// TwinCAT 3 PLC project Autoloader
// ProgramVersion: 3.1.4023.0
// libraries:
//   FESTO CMMT_AS Drive Control, * (Sensata Mech Sofia)
//   Motors_AFAG_CoE, * (Sensata Technologies Bulgaria)
//   Motors_DUTs, * (Sensata Technologies Bulgaria)
//   Tc2_Math, * (Beckhoff Automation GmbH)
//   Tc2_Standard, * (Beckhoff Automation GmbH)
//   Tc2_System, * (Beckhoff Automation GmbH)
//   Tc2_TcpIp, * (Beckhoff Automation GmbH)
//   Tc2_Utilities, * (Beckhoff Automation GmbH)
//   Tc3_Module, * (Beckhoff Automation GmbH)
//   Festo_PtP_Base,3.5.10.47,Festo
//   Festo_PtP_CiA402,3.5.10.47,Festo
//   Festo_PtP_CiA402_ETC,3.5.10.47,Festo
//   Festo_PtP_CiA402_ETC_CMMT_AS,3.5.10.47,Festo
//   Festo_PtP_Virtual,3.5.10.47,Festo
//   Tc3_LinMot,1.1.0.0,NTI AG
// project tree:
//   DUTs/ camResult.TcDUT, controlCommands.TcDUT, dataRequestCam.TcDUT, dataRequestRobot.TcDUT, E_RobotStates.TcDUT, imageIO.TcDUT, ioType.TcDUT, globalDeps.TcDUT, stationBase.TcDUT
//   DUTs/Stations/incComm/ incCommDisplayStates.TcDUT, incCommImage.TcDUT, incCommIO.TcDUT, incCommSettings.TcDUT, incCommStates.TcDUT
//   DUTs/Stations/inserterLoad/ inserterLoadDisplayStates.TcDUT, inserterLoadImage.TcDUT, inserterLoadIO.TcDUT, inserterLoadRecipe.TcDUT, inserterLoadSettings.TcDUT, inserterLoadStates.TcDUT
//   DUTs/Stations/inserterUnload/ inserterUnLoadImage.TcDUT, inserterUnLoadRecipe.TcDUT, inserterUnLoadDisplayStates.TcDUT, inserterUnLoadIO.TcDUT, inserterUnLoadSettings.TcDUT, inserterUnLoadStates.TcDUT
//   DUTs/Stations/machine/ machineDisplayStates.TcDUT, machineImage.TcDUT, machineIO.TcDUT, machineSettings.TcDUT, machineStates.TcDUT
//   DUTs/Stations/roboArm/ roboArmDisplayStates.TcDUT, roboArmImage.TcDUT, roboArmIO.TcDUT, roboArmSettings.TcDUT, roboArmsRecipe.TcDUT, roboArmStates.TcDUT
//   DUTs/Stations/stackerLoad/ palletParamsL.TcDUT, stackerLoadDisplayStates.TcDUT, stackerLoadImage.TcDUT, stackerLoadIO.TcDUT, stackerLoadSettings.TcDUT, stackerLoadStates.TcDUT
//   DUTs/Stations/stackerUnload/ palletParamsU.TcDUT, stackerUnLoadDisplayStates.TcDUT, stackerUnLoadImage.TcDUT, stackerUnLoadIO.TcDUT, stackerUnLoadSettings.TcDUT, stackerUnLoadStates.TcDUT
//   GVLs/ Consts.TcGVL, DEBUG.TcGVL, Global.TcGVL, Stations.TcGVL, TagsHMI.TcGVL, TagsRobot.TcGVL
//   / PlcTask.TcTTO, RobotTask.TcTTO
//   POUs/ MAIN.TcPOU, ROBOT.TcPOU, stateMachine.TcPOU, ioControl.TcPOU
//   POUs/Mitsubishi/DUT/Communication/PacketsStructure/Input/ ST_Robot_Mitsubishi_Packet_1000.TcDUT, ST_Robot_Mitsubishi_Packet_1100.TcDUT, ST_Robot_Mitsubishi_Packet_1101.TcDUT, ST_Robot_Mitsubishi_Packet_1102.TcDUT, ST_Robot_Mitsubishi_Packet_1103.TcDUT
//   POUs/Mitsubishi/DUT/Communication/PacketsStructure/Output/ ST_Robot_Mitsubishi_Packet_2000.TcDUT, ST_Robot_Mitsubishi_Packet_2010.TcDUT, ST_Robot_Mitsubishi_Packet_2011.TcDUT, ST_Robot_Mitsubishi_Packet_2012.TcDUT, ST_Robot_Mitsubishi_Packet_2013.TcDUT, ST_Robot_Mitsubishi_Packet_2014.TcDUT, ST_Robot_Mitsubishi_Packet_2015.TcDUT, ST_Robot_Mitsubishi_Packet_2016.TcDUT, ST_Robot_Mitsubishi_Packet_2017.TcDUT, ST_Robot_Mitsubishi_Packet_2018.TcDUT, ST_Robot_Mitsubishi_Packet_2019.TcDUT, ST_Robot_Mitsubishi_Packet_2100.TcDUT, ST_Robot_Mitsubishi_Packet_2101.TcDUT
//   POUs/Mitsubishi/DUT/Communication/ ST_Robot_Misubishi_Packet_Manager.TcDUT
//   POUs/Mitsubishi/DUT/ E_Communication_Send_States.TcDUT, E_Robot_Mitsubishi_States.TcDUT, ST_Robot_Mitsubishi.TcDUT
//   POUs/Mitsubishi/ FB_Robot_Mitsubishi.TcPOU, FB_Robot_Mitsubishi_ReceivePacket.TcPOU, FB_Robot_Mitsubishi_SendPacket.TcPOU
//   POUs/Mitsubishi/Func/ FB_EXTRACT_HEX_AND_FLIP.TcPOU, FB_HEXSTR_TO_DINT.TcPOU
//   POUs/Mitsubishi/Sub/ FB_ClearOutputBuffer.TcPOU, FB_SetOutputBuffer.TcPOU
//   POUs/Stations/ incCommStation.TcPOU, insertLoadStation.TcPOU, insertUnloadStation.TcPOU, machineStation.TcPOU, roboArmStation.TcPOU, stackerLoadStation.TcPOU, stackerUnloadStation.TcPOU
// real-time tasks:
//   TASK PlcTask: cycle T#10ms, priority 20, ADS port 350
//   TASK RobotTask: cycle T#10ms, priority 1, ADS port 351
// I/O:
//   DEVICE Device 1 (EtherCAT), AmsNetId 169.254.245.124.2.1
//     Term 1 (EK1100) [EK1100 EtherCAT Coupler (2A E-Bus)]
//       Term 2 (EL1008) [EL1008 8Ch. Dig. Input 24V, 3ms]
//       Term 3 (EL1008) [EL1008 8Ch. Dig. Input 24V, 3ms]
//       Term 4 (EL1008) [EL1008 8Ch. Dig. Input 24V, 3ms]
//       Term 5 (EL2808) [EL2808 8Ch. Dig. Output 24V, 0.5A]
//       Term 6 (EL2808) [EL2808 8Ch. Dig. Output 24V, 0.5A]
//       Term 7 (EL2808) [EL2808 8Ch. Dig. Output 24V, 0.5A]
//       Term 8 (EK1310) [EK1310 EtherCAT P extension with feed-in]
//     Box 9 (EPP2316-0003) [EPP2316-0003 8 Ch. Dig. In, 10µs, 8Ch. Dig. Out 24V, 0,5A, Diagnostic, 10-Pole Plug Connector]
//     Box 10 (EPP2316-0003) [EPP2316-0003 8 Ch. Dig. In, 10µs, 8Ch. Dig. Out 24V, 0,5A, Diagnostic, 10-Pole Plug Connector]
//     Box 11 (CMMT-AS) [CMMT-AS]
//     Box 12 (CMMT-AS) [CMMT-AS]
//     Box 13 (C1150-EC-XC-1S) [C1150-EC-XC-1S V1.7b5]
//     Box 14 (C1150-EC-XC-1S) [C1150-EC-XC-1S V1.7b5]
//     Box 15 (EX260-SEC1) [EX260-SEC1 EtherCAT SI Unit (32DO_PNP) Rev1.2]
//     Box 16 (EP1008-0001) [EP1008-0001 8 Ch. Dig. Input 24V, 3ms, M8]
//     Box 17 (EP1008-0001) [EP1008-0001 8 Ch. Dig. Input 24V, 3ms, M8]
//     Box 18 (EP1008-0001) [EP1008-0001 8 Ch. Dig. Input 24V, 3ms, M8]
// variable links:
//   Autoloader/Autoloader Instance <-> Device 1 (EtherCAT)/Box 10 (EPP2316-0003)
//     PlcTask Inputs/Global.INPUT_IMAGE[10] <-> DIG Inputs/Input 1
//     PlcTask Inputs/Global.INPUT_IMAGE[10] @bit {1..7} <-> DIG Inputs/Input {2..8}  (7 links)
//     PlcTask Outputs/Global.OUTPUT_IMAGE[10] <-> DIG Outputs/Output 1
//     PlcTask Outputs/Global.OUTPUT_IMAGE[10] @bit {1..7} <-> DIG Outputs/Output {2..8}  (7 links)
//   Autoloader/Autoloader Instance <-> Device 1 (EtherCAT)/Box 11 (CMMT-AS)
//     PlcTask Inputs/Stations.sLoadAxis.AdsAddr_In <-> InfoData/AdsAddr
//     PlcTask Inputs/Stations.sLoadAxis.ModesOfOperationDisplay_In <-> Inputs/Modes of operation display
//     PlcTask Inputs/Stations.sLoadAxis.PositionActualValue_In <-> Inputs/Position actual value
//     PlcTask Inputs/Stations.sLoadAxis.SlaveState_In <-> InfoData/State
//     PlcTask Inputs/Stations.sLoadAxis.Statusword_In <-> Inputs/Statusword
//     PlcTask Inputs/Stations.sLoadAxis.TorqueActualValue_In <-> Inputs/Torque actual value
//     PlcTask Inputs/Stations.sLoadAxis.VelocityActualValue_In <-> Inputs/Velocity actual value
//     PlcTask Inputs/Stations.sLoadAxis.WcState_In <-> WcState/WcState
//     PlcTask Outputs/Stations.sLoadAxis.Controlword_Out <-> Outputs/Controlword
//     PlcTask Outputs/Stations.sLoadAxis.ModesOfOperation_Out <-> Outputs/Modes of operation
//     PlcTask Outputs/Stations.sLoadAxis.ProfileVelocity_Out <-> Outputs/Profile velocity
//     PlcTask Outputs/Stations.sLoadAxis.TargetPosition_Out <-> Outputs/Target position
//     PlcTask Outputs/Stations.sLoadAxis.TargetTorque_Out <-> Outputs/Target torque
//     PlcTask Outputs/Stations.sLoadAxis.TargetVelocity_Out <-> Outputs/Target velocity
//   Autoloader/Autoloader Instance <-> Device 1 (EtherCAT)/Box 12 (CMMT-AS)
//     PlcTask Inputs/Stations.sUnloadAxis.AdsAddr_In <-> InfoData/AdsAddr
//     PlcTask Inputs/Stations.sUnloadAxis.ModesOfOperationDisplay_In <-> Inputs/Modes of operation display
//     PlcTask Inputs/Stations.sUnloadAxis.PositionActualValue_In <-> Inputs/Position actual value
//     PlcTask Inputs/Stations.sUnloadAxis.SlaveState_In <-> InfoData/State
//     PlcTask Inputs/Stations.sUnloadAxis.Statusword_In <-> Inputs/Statusword
//     PlcTask Inputs/Stations.sUnloadAxis.TorqueActualValue_In <-> Inputs/Torque actual value
//     PlcTask Inputs/Stations.sUnloadAxis.VelocityActualValue_In <-> Inputs/Velocity actual value
//     PlcTask Inputs/Stations.sUnloadAxis.WcState_In <-> WcState/WcState
//     PlcTask Outputs/Stations.sUnloadAxis.Controlword_Out <-> Outputs/Controlword
//     PlcTask Outputs/Stations.sUnloadAxis.ModesOfOperation_Out <-> Outputs/Modes of operation
//     PlcTask Outputs/Stations.sUnloadAxis.ProfileVelocity_Out <-> Outputs/Profile velocity
//     PlcTask Outputs/Stations.sUnloadAxis.TargetPosition_Out <-> Outputs/Target position
//     PlcTask Outputs/Stations.sUnloadAxis.TargetTorque_Out <-> Outputs/Target torque
//     PlcTask Outputs/Stations.sUnloadAxis.TargetVelocity_Out <-> Outputs/Target velocity
//   Autoloader/Autoloader Instance <-> Device 1 (EtherCAT)/Box 13 (C1150-EC-XC-1S)
//     PlcTask Inputs/Stations.insertLoadAxis.DrvToPlc/ComActualPosition <-> Default Inputs/ActualPosition
//     PlcTask Inputs/Stations.insertLoadAxis.DrvToPlc/ComDemandPosition <-> Default Inputs/DemandPosition
//     PlcTask Inputs/Stations.insertLoadAxis.DrvToPlc/StateVar <-> Default Inputs/StateVar
//     PlcTask Inputs/Stations.insertLoadAxis.DrvToPlc/StatusWord <-> Default Inputs/StatusWord
//     PlcTask Inputs/Stations.insertLoadAxis.DrvToPlc/WarnWord <-> Default Inputs/WarnWord
//     PlcTask Outputs/Stations.insertLoadAxis.PlcToDrv/ControlWord <-> Default Outputs/Control Word
//     PlcTask Outputs/Stations.insertLoadAxis.PlcToDrv/MCHeader <-> Default Outputs/Motion Command Header
//     PlcTask Outputs/Stations.insertLoadAxis.PlcToDrv/MCParaDWord_00_03 <-> Default Outputs/Motion Command Par 1
//     PlcTask Outputs/Stations.insertLoadAxis.PlcToDrv/MCParaDWord_04_07 <-> Default Outputs/Motion Command Par 2
//     PlcTask Outputs/Stations.insertLoadAxis.PlcToDrv/MCParaDWord_08_11 <-> Default Outputs/Motion Command Par 3
//     PlcTask Outputs/Stations.insertLoadAxis.PlcToDrv/MCParaDWord_12_15 <-> Default Outputs/Motion Command Par 4
//     PlcTask Outputs/Stations.insertLoadAxis.PlcToDrv/MCParaDWord_16_19 <-> Default Outputs/Motion Command Par 5
//   Autoloader/Autoloader Instance <-> Device 1 (EtherCAT)/Box 14 (C1150-EC-XC-1S)
//     PlcTask Inputs/Stations.insertUnLoadAxis.DrvToPlc/ComActualPosition <-> Default Inputs/ActualPosition
//     PlcTask Inputs/Stations.insertUnLoadAxis.DrvToPlc/ComDemandPosition <-> Default Inputs/DemandPosition
//     PlcTask Inputs/Stations.insertUnLoadAxis.DrvToPlc/StateVar <-> Default Inputs/StateVar
//     PlcTask Inputs/Stations.insertUnLoadAxis.DrvToPlc/StatusWord <-> Default Inputs/StatusWord
//     PlcTask Inputs/Stations.insertUnLoadAxis.DrvToPlc/WarnWord <-> Default Inputs/WarnWord
//     PlcTask Outputs/Stations.insertUnLoadAxis.PlcToDrv/ControlWord <-> Default Outputs/Control Word
//     PlcTask Outputs/Stations.insertUnLoadAxis.PlcToDrv/MCHeader <-> Default Outputs/Motion Command Header
//     PlcTask Outputs/Stations.insertUnLoadAxis.PlcToDrv/MCParaDWord_00_03 <-> Default Outputs/Motion Command Par 1
//     PlcTask Outputs/Stations.insertUnLoadAxis.PlcToDrv/MCParaDWord_04_07 <-> Default Outputs/Motion Command Par 2
//     PlcTask Outputs/Stations.insertUnLoadAxis.PlcToDrv/MCParaDWord_08_11 <-> Default Outputs/Motion Command Par 3
//     PlcTask Outputs/Stations.insertUnLoadAxis.PlcToDrv/MCParaDWord_12_15 <-> Default Outputs/Motion Command Par 4
//     PlcTask Outputs/Stations.insertUnLoadAxis.PlcToDrv/MCParaDWord_16_19 <-> Default Outputs/Motion Command Par 5
//   Autoloader/Autoloader Instance <-> Device 1 (EtherCAT)/Box 15 (EX260-SEC1)
//     PlcTask Outputs/Global.OUTPUT_IMAGE[150] <-> Byte 0/Output
//     PlcTask Outputs/Global.OUTPUT_IMAGE[151] <-> Byte 1/Output
//     PlcTask Outputs/Global.OUTPUT_IMAGE[152] <-> Byte 2/Output
//   Autoloader/Autoloader Instance <-> Device 1 (EtherCAT)/Box 16 (EP1008-0001)
//     PlcTask Inputs/Global.INPUT_IMAGE[16] <-> Channel 1/Input
//     PlcTask Inputs/Global.INPUT_IMAGE[16] @bit {1..7} <-> Channel {2..8}/Input  (7 links)
//   Autoloader/Autoloader Instance <-> Device 1 (EtherCAT)/Box 17 (EP1008-0001)
//     PlcTask Inputs/Global.INPUT_IMAGE[17] <-> Channel 1/Input
//     PlcTask Inputs/Global.INPUT_IMAGE[17] @bit {1..7} <-> Channel {2..8}/Input  (7 links)
//   Autoloader/Autoloader Instance <-> Device 1 (EtherCAT)/Box 18 (EP1008-0001)
//     PlcTask Inputs/Global.INPUT_IMAGE[18] <-> Channel 1/Input
//     PlcTask Inputs/Global.INPUT_IMAGE[18] @bit {1..7} <-> Channel {2..8}/Input  (7 links)
//   Autoloader/Autoloader Instance <-> Device 1 (EtherCAT)/Box 9 (EPP2316-0003)
//     PlcTask Inputs/Global.INPUT_IMAGE[9] <-> DIG Inputs/Input 1
//     PlcTask Inputs/Global.INPUT_IMAGE[9] @bit {1..7} <-> DIG Inputs/Input {2..8}  (7 links)
//     PlcTask Outputs/Global.OUTPUT_IMAGE[9] <-> DIG Outputs/Output 1
//     PlcTask Outputs/Global.OUTPUT_IMAGE[9] @bit {1..7} <-> DIG Outputs/Output {2..8}  (7 links)
//   Autoloader/Autoloader Instance <-> Device 1 (EtherCAT)/Term 1 (EK1100)/Term 2 (EL1008)
//     PlcTask Inputs/Global.INPUT_IMAGE[2] <-> Channel 1/Input
//     PlcTask Inputs/Global.INPUT_IMAGE[2] @bit {1..7} <-> Channel {2..8}/Input  (7 links)
//   Autoloader/Autoloader Instance <-> Device 1 (EtherCAT)/Term 1 (EK1100)/Term 3 (EL1008)
//     PlcTask Inputs/Global.INPUT_IMAGE[3] <-> Channel 1/Input
//     PlcTask Inputs/Global.INPUT_IMAGE[3] @bit {1..7} <-> Channel {2..8}/Input  (7 links)
//   Autoloader/Autoloader Instance <-> Device 1 (EtherCAT)/Term 1 (EK1100)/Term 4 (EL1008)
//     PlcTask Inputs/Global.INPUT_IMAGE[4] <-> Channel 1/Input
//     PlcTask Inputs/Global.INPUT_IMAGE[4] @bit {1..7} <-> Channel {2..8}/Input  (7 links)
//   Autoloader/Autoloader Instance <-> Device 1 (EtherCAT)/Term 1 (EK1100)/Term 5 (EL2808)
//     PlcTask Outputs/Global.OUTPUT_IMAGE[5] <-> Channel 1/Output
//     PlcTask Outputs/Global.OUTPUT_IMAGE[5] @bit {1..7} <-> Channel {2..8}/Output  (7 links)
//   Autoloader/Autoloader Instance <-> Device 1 (EtherCAT)/Term 1 (EK1100)/Term 6 (EL2808)
//     PlcTask Outputs/Global.OUTPUT_IMAGE[6] <-> Channel 1/Output
//     PlcTask Outputs/Global.OUTPUT_IMAGE[6] @bit {1..7} <-> Channel {2..8}/Output  (7 links)
//   Autoloader/Autoloader Instance <-> Device 1 (EtherCAT)/Term 1 (EK1100)/Term 7 (EL2808)
//     PlcTask Outputs/Global.OUTPUT_IMAGE[7] <-> Channel 1/Output
//     PlcTask Outputs/Global.OUTPUT_IMAGE[7] @bit {1..7} <-> Channel {2..8}/Output  (7 links)

CONFIGURATION Autoloader
    RESOURCE PLC ON TwinCAT3
        TASK PlcTask(INTERVAL := T#10ms, PRIORITY := 20);
        TASK RobotTask(INTERVAL := T#10ms, PRIORITY := 1);
        PROGRAM MAIN WITH PlcTask : MAIN;
        PROGRAM Robot WITH RobotTask : Robot;
    END_RESOURCE
END_CONFIGURATION

// ---- DUTs/camResult.TcDUT
{attribute 'qualified_only'}

TYPE camResult :
(
	null          := 0,                         // Неправилен резултат от камерата
	turnCCW,
	turnCW
	
)DINT;
END_TYPE

// ---- DUTs/controlCommands.TcDUT
{attribute 'qualified_only'}

// Команди който идват от I&C

TYPE controlCommands :
(
	null		:= 0,
	stop,
	start
	
)DINT;
END_TYPE

// ---- DUTs/dataRequestCam.TcDUT
{attribute 'qualified_only'}




TYPE dataRequestCam :
(
	done               := Consts.NO_REQUEST,
	error              := Consts.REQUEST_ERROR,
	
	camShotRecipe1     := 1,           // Тази стойност НЕ трябва да се променя - винаги е 1 !
	camShotRecipe2,
	camShotRecipe3,
	camShotRecipe4,
	camShotRecipe5,
	camShotRecipe6,
	camShotRecipe7,
	camShotRecipe8,
	camShotRecipe9,
	camShotRecipe10,
	camShotRecipe11,
	camShotRecipe12,
	camShotRecipe13,
	camShotRecipe14,
	camShotRecipe15
	
	
)DINT;
END_TYPE

// ---- DUTs/dataRequestRobot.TcDUT
{attribute 'qualified_only'}


TYPE dataRequestRobot :
(
	

	done       := Consts.NO_REQUEST,
	error      := Consts.REQUEST_ERROR,
	
	roboInit	   := 100,				// Зарежда MAINPROGRAM и изчаква робота да е в READY
	
	roboPrg_Home   := 1,
	roboPrg_SensorLoad,
	roboPrg_SensorUnload,
	roboPrg_SensorDown,
	roboPrg_PreLoad,
	roboPrg_Load,
	roboPrg_PreUnload,
	roboPrg_Unload,
	roboPrg_LoadStacker,
	roboPrg_UnloadStacker,
	roboPrg_EmptyPlace,
	roboPrg_HomeWithPallet
	
)DINT;
END_TYPE

// ---- DUTs/E_RobotStates.TcDUT
{attribute 'qualified_only'}
{attribute 'to_string'}
TYPE E_RobotStates :
(
	STATE_WAITING_FOR_INIT := 0,
	STATE_INIT_ROBOT_TOGGLE,
	STATE_INIT_ROBOT_ON,
	STATE_INIT_CHECK_ROBOT_ERROR,
	STATE_INIT_CHECK_ROBOT_ERROR_DONE,
	STATE_INIT_CHECK_ROBOT_READY,
	STATE_INIT_CHECK_ROBOT_READY_DONE,
	STATE_INIT_CHECK_ROBOT_SERVOON,
	STATE_INIT_CHECK_ROBOT_SERVOON_DONE,
	STATE_INIT_DONE,
	STATE_WAITING_FOR_COMMAND := 100,
	STATE_WAITING_START_PRG,
	STATE_PROGRAM_DONE,	//Ready
	STATE_ERROR := 1000	// Default error
) UDINT;
END_TYPE

// ---- DUTs/imageIO.TcDUT
TYPE imageIO :
STRUCT
	
	// Това е структура която "вързва" даден сигнал от stataionIO с опеделен такъв от В/И image на TC
	// Идеята е да не се мисли за обновяване на сигналите, т.е. да няма копиране на няколко места за да се обнови статуса им.
	// TO DO -> да се реализира подхода и за аналогови сигнали 
	
	stIO			: REFERENCE TO BOOL; 						                // име на сигнал от stationIO
	image			: POINTER TO ARRAY [0..Consts.MAX_IO_POINTS] OF BYTE;       // масив на IO image
	iType           : ioType; 													// тип
	iByte 			: UINT;                                                     // номер на байт от масива
	iBit			: UINT; 									                // номер на бит от байта
	 
END_STRUCT
END_TYPE

// ---- DUTs/ioType.TcDUT
{attribute 'qualified_only'}

// Опеределя вида на перифериятя - за сега е само входе и изходен бит

TYPE ioType :
(
	INPUT_BIT   := 1,
	OUTPUT_BIT
)DINT;
END_TYPE

// ---- DUTs/globalDeps.TcDUT
{attribute 'qualified_only'}

TYPE globalDeps :
(
	
	// За machine station
	depMachineInitDone 			:=    10,
	depMachineAuto,
	depMachineStopping, 
	depMachineStop,
	depMachinePurgeStart,
	depMachinePurgeRobot,
	depMacinePurgeStackers,

	// За staker load station
	depSLoadInit,
	depSLoadWaitRobotReady,
	depSLoadRobotOutOfReach,
	depSLoadStop,
	depSLoadPurgeDone,
	depSLoadRobotLoadGrip,
	depSLoadStationReady,
	depSLoadStationDone,
	
	// За staker unload station
	depSUnloadInit,
	depSUnloadStop,
	depSUnloadWaitRobotReady,
	depSUnloadRobotUnloadGrip,
	depSUnloadRobotOutOfReach,	
	depSUnloadPurgeDone,
	depSUnloadStationReady,
	
	// За Inc Comm station
	depIncCommModeDone,
	depIncIncComm,
	depIncCycleDone,
	depIncStop,
	depIncPurgeDone,
	
	// За RoboArm station
	depRoboInitDone,
	depRoboStop,
	depRoboLoadPalletUnlock,
	depRoboUnLoadPalletLock,
	depRoboUnLodPalletFull,
	depRoboPurgeDone,
	depRoboGripOpen,
	depRoboGripClose,
	depRoboILoadOnPos,
	depRoboULoadOnPos,
	depRoboLoadSensor,
	depRoboStartLoadStacker,
	depRobotClearUnLoadStacker,
	
	// За inserter load station
	depILoadInitDone,
    depILoadWaitRobotReady,	
	depILoadRobotBack,
	depILoadSignalForLoad,
	depILoadWaitIndex,
	depILoadDone,
	depILoadStop,
	
	// За inserter unload station
	depULoadInitDone,
    depULoadWaitRobotReady,	
	depULoadWaitIndex,
	depULoadDone,
	depULoadRobotOutOfRich,	
	depULoadStop
	
)DINT;
END_TYPE

// ---- DUTs/Stations/incComm/incCommDisplayStates.TcDUT
{attribute 'qualified_only'}

TYPE incCommDisplayStates :
(
	
	dStStartingUp   := 10,
	dStStandBy,
	dStIncModeSignalsError,
	dStWaitForAllStatinsReady,
	dStDialTableIndexPermition,
	dStDialTableIndexReady,
	dStStationIsStopped,
	dStWaitForNextStep
	
	
	
)DINT;
END_TYPE

// ---- DUTs/Stations/incComm/incCommImage.TcDUT
TYPE incCommImage :
STRUCT
	
	// Входове
    xSignalStop 		: imageIO := ( stIO   := Stations.incCommHmiIO.x_SignalStop,
									   image  := ADR(Global.INPUT_IMAGE),
									   iType  := ioType.INPUT_BIT,
									   iByte  := 4,
									   iBit   := 0 );	
									   
    xSignalStart 		: imageIO := ( stIO   := Stations.incCommHmiIO.x_SignalStart,
									   image  := ADR(Global.INPUT_IMAGE),
									   iType  := ioType.INPUT_BIT,
									   iByte  := 4,
									   iBit   := 1 );

    xPickNestLoaded 	: imageIO := ( stIO   := Stations.incCommHmiIO.x_pickNestLoaded,
									   image  := ADR(Global.INPUT_IMAGE),
									   iType  := ioType.INPUT_BIT,
									   iByte  := 4,
									   iBit   := 2 );
									   
    xDailIndexDone 	: imageIO := ( stIO   := Stations.incCommHmiIO.x_DailIndexDone,
									   image  := ADR(Global.INPUT_IMAGE),
									   iType  := ioType.INPUT_BIT,
									   iByte  := 4,
									   iBit   := 3);									   

    xRecipeBit0 	    : imageIO := ( stIO   := Stations.incCommHmiIO.x_recipeBit0,
									   image  := ADR(Global.INPUT_IMAGE),
									   iType  := ioType.INPUT_BIT,
									   iByte  := 4,
									   iBit   := 4);

    xRecipeBit1 	    : imageIO := ( stIO   := Stations.incCommHmiIO.x_recipeBit1,
									   image  := ADR(Global.INPUT_IMAGE),
									   iType  := ioType.INPUT_BIT,
									   iByte  := 4,
									   iBit   := 5);	
									   
   xRecipeBit2 	    	: imageIO := ( stIO   := Stations.incCommHmiIO.x_recipeBit2,
									   image  := ADR(Global.INPUT_IMAGE),
									   iType  := ioType.INPUT_BIT,
									   iByte  := 4,
									   iBit   := 6);

   xRecipeBit3 	    	: imageIO := ( stIO   := Stations.incCommHmiIO.x_recipeBit3,
									   image  := ADR(Global.INPUT_IMAGE),
									   iType  := ioType.INPUT_BIT,
									   iByte  := 4,
									   iBit   := 7);									   
									   									   

	// Изходи
    yProductChange 		: imageIO := ( stIO   := Stations.incCommHmiIO.y_productChange,
									   image  := ADR(Global.OUTPUT_IMAGE),
									   iType  := ioType.OUTPUT_BIT,
									   iByte  := 5,
									   iBit   := 0 );

    yAlarm 		        : imageIO := ( stIO   := Stations.incCommHmiIO.y_alarm,
									   image  := ADR(Global.OUTPUT_IMAGE),
									   iType  := ioType.OUTPUT_BIT,
									   iByte  := 5,
									   iBit   := 1 );

    yDailIndex 		    : imageIO := ( stIO   := Stations.incCommHmiIO.y_dailIndex,
									   image  := ADR(Global.OUTPUT_IMAGE),
									   iType  := ioType.OUTPUT_BIT,
									   iByte  := 5,
									   iBit   := 2 );	
					   	

END_STRUCT
END_TYPE

// ---- DUTs/Stations/incComm/incCommIO.TcDUT
TYPE incCommIO :
STRUCT
	
	// Входове
	x_SignalStop			: BOOL; 						// Стоп бутон на InC
	x_SignalStart			: BOOL; 						// Старт бутон на InC
	x_pickNestLoaded        : BOOL; 						// Има готова бройка за взимане 						// Може да се остави бройка - гнездото е празно
	x_recipeBit0			: BOOL; 						// Режим на работа HEX24
    x_recipeBit1			: BOOL;							// Режим на работа HEX27
	x_recipeBit2            : BOOL;
	x_recipeBit3            : BOOL;
	x_dailIndexDone			: BOOL;							// Индекс масата е направила един ход - движението е завършено       
	
	// Изходи
	y_productChange			: BOOL;                         // InC има разрешение да стартира нов лот (и да смени продукта HEX24 или HEX27)
	y_alarm					: BOOL; 						// Има активна аларма
	y_dailIndex				: BOOL; 						// InC е безопастно да завърти индекс масата с един ход

END_STRUCT
END_TYPE

// ---- DUTs/Stations/incComm/incCommSettings.TcDUT
TYPE incCommSettings :
STRUCT
END_STRUCT
END_TYPE

// ---- DUTs/Stations/incComm/incCommStates.TcDUT
{attribute 'qualified_only'}

TYPE incCommStates :
(
		stNull      :=    Consts.ST_NULL,
		stStartUp   :=    Consts.ST_START_UP,
		stInit      :=    Consts.ST_INIT,
		stReady     :=    Consts.ST_READY,
		stStop      :=    Consts.ST_STOP,
		stStepBlock :=    Consts.ST_STEP_BLOCK,	
		stEMG		:=    Consts.ST_EMG,
		
		
		stSetMode                := 1000,
		stStationStop,
		
		stIndexStart,
		stIndexEnableStations,
		stIndexStationsReady,
		stSignalStations,		
		stIndexEnable, 
		stIndexReady,
		stIndexCheck, 
		stIndexDone,
		
		stPurgeStart,
		stPurgeFinish,
		stPurgeDone,

		stErrCommFault

)DINT;
END_TYPE

// ---- DUTs/Stations/inserterLoad/inserterLoadDisplayStates.TcDUT
{attribute 'qualified_only'}

TYPE inserterLoadDisplayStates :
(
	
	dStStartUp,
	dStStandBy,
	dStStationIsStopped,
	dStStationIsReseting,
	dStWorking,
	dStStationReady,
	dStWaitForNextStep,
	
	dStGripperDidNotClose,
	dStGripperDidNotOpen,
	dStInserterDidNotMoveDown,
	dStInserterDidNotMoveUp,
	dStDriveDidNotHome,
	dStDriveTimeOutMove,
	dStDriveError,
	dStCameraTimeOut,
	dStCameraError,
	dStCameraBadResult,
	dStInitSensorGripError
	
	
)DINT;
END_TYPE

// ---- DUTs/Stations/inserterLoad/inserterLoadImage.TcDUT
TYPE inserterLoadImage :
STRUCT
	
   // Входове
   xGrip_open 	        : imageIO := ( stIO   := Stations.insertLoadHmiIO.x_Grip_open,
									   image  := ADR(Global.INPUT_IMAGE),
									   iType  := ioType.INPUT_BIT,
									   iByte  := 18,
									   iBit   := 0 );	
									   
   xGrip_close			: imageIO := ( stIO   := Stations.insertLoadHmiIO.x_Grip_close,
									   image  := ADR(Global.INPUT_IMAGE),
									   iType  := ioType.INPUT_BIT,
									   iByte  := 18,
									   iBit   := 1 );

    xInsert_up 			: imageIO := ( stIO   := Stations.insertLoadHmiIO.x_Insert_up,
									   image  := ADR(Global.INPUT_IMAGE),
									   iType  := ioType.INPUT_BIT,
									   iByte  := 18,
									   iBit   := 2 );
									   
    xInsert_down 		: imageIO := ( stIO   := Stations.insertLoadHmiIO.x_Insert_down,
									   image  := ADR(Global.INPUT_IMAGE),
									   iType  := ioType.INPUT_BIT,
									   iByte  := 18,
									   iBit   := 3 );									   	   
									   
    xNest 			    : imageIO := ( stIO   := Stations.insertLoadHmiIO.x_Nest,
									   image  := ADR(Global.INPUT_IMAGE),
									   iType  := ioType.INPUT_BIT,
									   iByte  := 3,
									   iBit   := 0 );

	// Изходи								   									   
    yGrip_open 			: imageIO := ( stIO   := Stations.insertLoadHmiIO.y_Grip_open,
									   image  := ADR(Global.OUTPUT_IMAGE),
									   iType  := ioType.OUTPUT_BIT,
									   iByte  := 150,
									   iBit   := 0 ); 

    yGrip_close 		: imageIO := ( stIO   := Stations.insertLoadHmiIO.y_Grip_close,
									   image  := ADR(Global.OUTPUT_IMAGE),
									   iType  := ioType.OUTPUT_BIT,
									   iByte  := 150,
									   iBit   := 1 ); 

    yInsert_up 			: imageIO := ( stIO   := Stations.insertLoadHmiIO.y_Insert_up,
									   image  := ADR(Global.OUTPUT_IMAGE),
									   iType  := ioType.OUTPUT_BIT,
									   iByte  := 150,
									   iBit   := 5 ); 

    yInsert_down 		: imageIO := ( stIO   := Stations.insertLoadHmiIO.y_Insert_down,
									   image  := ADR(Global.OUTPUT_IMAGE),
									   iType  := ioType.OUTPUT_BIT,
									   iByte  := 150,
									   iBit   := 4 ); 	
									   
    yFlashLight 		: imageIO := ( stIO   := Stations.insertLoadHmiIO.y_FlashLight,
									   image  := ADR(Global.OUTPUT_IMAGE),
									   iType  := ioType.OUTPUT_BIT,
									   iByte  := 6,
									   iBit   := 4 ); 									   

	
  
END_STRUCT
END_TYPE

// ---- DUTs/Stations/inserterLoad/inserterLoadIO.TcDUT
TYPE inserterLoadIO :
STRUCT
	
	// Входове
	x_Grip_open				: BOOL;           // Грипера е отворен - сензор на цилиндър
    x_Grip_close            : BOOL;           // Грипера е затворен - сензор на цилиндър
	x_Insert_up             : BOOL;           // Инсъртъра е вдигнат - сензор на цилиндър
	x_Insert_down           : BOOL;           // Инсъртъра е свален	- сензор на цилиндър
	x_Nest                  : BOOL;           // Лазърен сензор - детектва имали продукт в гнездото под инсъртъра
	
	// Изходи
	y_Grip_open				: BOOL;           // Грипера е отворен -  цилиндър
    y_Grip_close            : BOOL;           // Грипера е затворен -  цилиндър
	y_Insert_up             : BOOL;           // Инсъртъра е вдигнат - цилиндър
	y_Insert_down           : BOOL;           // Инсъртъра е свален	-  цилиндър
	y_FlashLight            : BOOL;


END_STRUCT
END_TYPE

// ---- DUTs/Stations/inserterLoad/inserterLoadRecipe.TcDUT
TYPE inserterLoadRecipe :
STRUCT
	

	initRot               :   REAL   := 10;        // начало ротиране на грипера
	beforeGripRot         :   REAL   := 10;        // ротация преди да затвори грипера
	camRot 	              :   REAL   := 10;        // позиция на снимане
	cwRot                 :   REAL   := 10;        // завъртане на ccw след команда от камерата 
	ccwRot                :   REAL   := 10;        // завъртане на ccw след команда от камерата 



END_STRUCT
END_TYPE

// ---- DUTs/Stations/inserterLoad/inserterLoadSettings.TcDUT
TYPE inserterLoadSettings :
STRUCT
	
	axisWorkSpeed             :	  REAL   := 2000; 	   // скорост 
	axisAcc					  :   REAL   := 2;         // ускр.
	axisPres                  :   REAL   := 0.1;       // точност на позициониране
	rotParams                 :   ARRAY[1..Consts.MAX_RECIPE] OF inserterLoadRecipe; 	

END_STRUCT
END_TYPE

// ---- DUTs/Stations/inserterLoad/inserterLoadStates.TcDUT
{attribute 'qualified_only'}

TYPE inserterLoadStates :
(
		stNull      :=    Consts.ST_NULL,
		stStartUp   :=    Consts.ST_START_UP,
		stInit      :=    Consts.ST_INIT,
		stReady     :=    Consts.ST_READY,
		stStop      :=    Consts.ST_STOP,
		stStepBlock :=    Consts.ST_STEP_BLOCK,	
		stEMG		:=    Consts.ST_EMG,
		
		
		stPowerUp    :=    1000,
		stInitDone,
		stInserterLoadStopped,
		
		stResetStart,
		stResetSyncRobot,
		stResetGripOpen,
		stResetGripCheck,
		stResetMoveUpCheck,
		stResetLimitsCalc,		
		stResetDriveHome,
		stResetDriveCheck1,
		stResetDriveMove,
		stResetDriveCheck2,
		stResetDone,
		
		stPrepareStart,
		stPrepareNestCheck,
		stPrepareRobotWait,
		stPrepareDone,
		
		stLoadStart,
		stLoadDriveOn,
		stLoadDriveMove,
		stLoadDriveCheck,
		stLoadGripCheck,
		stLoadRobotSync,
		stLoadDone,
		
		stRotStart,
		stRotGripCheck,
		stRotDriveOn,
		stRotDriveMove,
		stRotDriveCheck,
		stRotCamShot,
		stRotCamCheck,
		stRotDone,
		
		stPosStart,
		stPosGripCheck,
		stPosDriveOn,
		stPosDriveMove,
		stPosDriveCheck,		
		stPosDone,
		
		stInsertStart,
		stInsertGripCheck,
		stInsertNestCheck,
		stInsertMoveDownCheck,
		stInsetDone,
		
		stReleaseStart,
		stReleaseGripCheck,
		stReleaseMoveUpCheck,
		stReleaseDriveOn,
		stReleaseDriveMove,
		stReleaseDriveCheck,
		stReleaseDone,
		
		stSyncIndexStart,
		stSyncIndexDone,
		
		
		stErrGripNotOpen,
		stErrGripNotClose,
		stErrInsertNotDown,
		stErrInsertNotUp,
		stErrDriveErr,
		stErrDriveTimeOut,
		stErrDriveHome,
		stErrCamTimeout,
		stErrCamErr,
		stErrCamBadResult,
		stErrInitSensor

)DINT;
END_TYPE

// ---- DUTs/Stations/inserterUnload/inserterUnLoadImage.TcDUT
TYPE inserterUnLoadImage :
STRUCT
	
 // Входове
   xGrip_open 	        : imageIO := ( stIO   := Stations.insertUnloadHmiIO.x_Grip_open,
									   image  := ADR(Global.INPUT_IMAGE),
									   iType  := ioType.INPUT_BIT,
									   iByte  := 18,
									   iBit   := 4 );	
									   
   xGrip_close			: imageIO := ( stIO   := Stations.insertUnloadHmiIO.x_Grip_close,
									   image  := ADR(Global.INPUT_IMAGE),
									   iType  := ioType.INPUT_BIT,
									   iByte  := 18,
									   iBit   := 5 );

    xInsert_up 			: imageIO := ( stIO   := Stations.insertUnloadHmiIO.x_Insert_up,
									   image  := ADR(Global.INPUT_IMAGE),
									   iType  := ioType.INPUT_BIT,
									   iByte  := 18,
									   iBit   := 6 );
									   
    xInsert_down 		: imageIO := ( stIO   := Stations.insertUnloadHmiIO.x_Insert_down,
									   image  := ADR(Global.INPUT_IMAGE),
									   iType  := ioType.INPUT_BIT,
									   iByte  := 18,
									   iBit   := 7 );									   	   
									   
    xNest 			    : imageIO := ( stIO   := Stations.insertUnloadHmiIO.x_Nest,
									   image  := ADR(Global.INPUT_IMAGE),
									   iType  := ioType.INPUT_BIT,
									   iByte  := 3,
									   iBit   := 1 );

	// Изходи								   									   
    yGrip_open 			: imageIO := ( stIO   := Stations.insertUnloadHmiIO.y_Grip_open,
									   image  := ADR(Global.OUTPUT_IMAGE),
									   iType  := ioType.OUTPUT_BIT,
									   iByte  := 150,
									   iBit   := 2 ); 

    yGrip_close 		: imageIO := ( stIO   := Stations.insertUnloadHmiIO.y_Grip_close,
									   image  := ADR(Global.OUTPUT_IMAGE),
									   iType  := ioType.OUTPUT_BIT,
									   iByte  := 150,
									   iBit   := 3 ); 

    yInsert_up 			: imageIO := ( stIO   := Stations.insertUnloadHmiIO.y_Insert_up,
									   image  := ADR(Global.OUTPUT_IMAGE),
									   iType  := ioType.OUTPUT_BIT,
									   iByte  := 150,
									   iBit   := 7 ); 

    yInsert_down 		: imageIO := ( stIO   := Stations.insertUnloadHmiIO.y_Insert_down,
									   image  := ADR(Global.OUTPUT_IMAGE),
									   iType  := ioType.OUTPUT_BIT,
									   iByte  := 150,
									   iBit   := 6 ); 	

	  

END_STRUCT
END_TYPE

// ---- DUTs/Stations/inserterUnload/inserterUnLoadRecipe.TcDUT
TYPE inserterUnLoadRecipe :
STRUCT
	

	initRot               :   REAL   := 10;        // начало ротиране на грипера
	workRot 	          :   REAL   := 10;        // позиция на вземане от робота
	afterOpenRot		  :   REAL   := 10;        // ротация след като отвори грипера, преди да се "извади" робота
 



END_STRUCT
END_TYPE

// ---- DUTs/Stations/inserterUnload/inserterUnLoadDisplayStates.TcDUT
{attribute 'qualified_only'}

TYPE inserterUnLoadDisplayStates :
(
	dStStartUp,
	dStStandBy,
	dStStationIsStopped,
	dStStationIsReseting,
	dStWorking,
	dStStationReady,
	dStWaitForNextStep,

	dStGripperDidNotClose,
	dStGripperDidNotOpen,
	dStInserterDidNotMoveDown,
	dStInserterDidNotMoveUp,
	dStDriveDidNotHome,
	dStDriveTimeOutMove,
	dStDriveError,
	dStCameraTimeOut,
	dStCameraError,
	dStCameraBadResult,
	dStInitSensorGripError,
	dStNoSensorInNest
	
	
)DINT;
END_TYPE

// ---- DUTs/Stations/inserterUnload/inserterUnLoadIO.TcDUT
TYPE inserterUnLoadIO :
STRUCT
	
	// Входове
	x_Grip_open				: BOOL;           // Грипера е отворен - сензор на цилиндър
    x_Grip_close            : BOOL;           // Грипера е затворен - сензор на цилиндър
	x_Insert_up             : BOOL;           // Инсъртъра е вдигнат - сензор на цилиндър
	x_Insert_down           : BOOL;           // Инсъртъра е свален	- сензор на цилиндър
	x_Nest                  : BOOL;           // Лазърен сензор - детектва имали продукт в гнездото под инсъртъра
	
	// Изходи
	y_Grip_open				: BOOL;           // Грипера е отворен -  цилиндър
    y_Grip_close            : BOOL;           // Грипера е затворен -  цилиндър
	y_Insert_up             : BOOL;           // Инсъртъра е вдигнат - цилиндър
	y_Insert_down           : BOOL;           // Инсъртъра е свален	-  цилиндър

END_STRUCT
END_TYPE

// ---- DUTs/Stations/inserterUnload/inserterUnLoadSettings.TcDUT
TYPE inserterUnLoadSettings :
STRUCT
	
	axisWorkSpeed             :	  REAL   := 2000; 	   // скорост 
	axisAcc					  :   REAL   := 2;         // ускр.
	axisPres                  :   REAL   := 0.1;       // точност на позициониране
	rotParams                 :   ARRAY[1..Consts.MAX_RECIPE] OF inserterUnLoadRecipe; 

END_STRUCT
END_TYPE

// ---- DUTs/Stations/inserterUnload/inserterUnLoadStates.TcDUT
{attribute 'qualified_only'}

TYPE inserterUnLoadStates :
(
		stNull      :=    Consts.ST_NULL,
		stStartUp   :=    Consts.ST_START_UP,
		stInit      :=    Consts.ST_INIT,
		stReady     :=    Consts.ST_READY,
		stStop      :=    Consts.ST_STOP,
		stStepBlock :=    Consts.ST_STEP_BLOCK,	
		stEMG		:=    Consts.ST_EMG,
		
		stPowerUp    :=    1000,
		stInitDone,
		stInserterUnloadStopped,
		
		stResetStart,
		stResetSyncRobot,
		stResetGripOpen,
		stResetGripCheck,
		stResetMoveUpCheck,
		stResetLimitsCalc,		
		stResetDriveHome,
		stResetDriveCheck,
		stResetDone,
		
		stPrepareStart, 
		stPrepareGripCheck,
		stPrepareNestCheck,
		stPrepareDriveOn,
		stPrepareDriveMove,
		stPrepareDriveCheck,
		stPrepareDone, 
		
		stMoveDownStart, 
		stMoveDownGripCheck,
		stMoveDownCheck,
		stMoveDownDone,
		
		stUnloadSensorStart,
		stUnloadSensorGripCheck1,
		stUnloadSensorGripCheck2,
		stUnloadSensorMoveCheck,
		stUnloadSensorDone,  
		
		stPosStart,   
		stPosGripCheck,
		stPosDriveOn,
		stPosDriveMove,
		stPosDriveCheck,
		stPosDone,   
		
		stReleaseStart,
		stReleaseSyncRobot, 
		stReleaseGripOpen,
		stReleaseGripCheck,
		stReleaseDriveOn,
		stReleaseDriveMove,
		stReleaseDriveCheck,
		stReleaseLoadDone,
		stReleaseDone,
		
		stSyncIndexStart,
		stSyncIndexDone,
		
		
		stErrGripNotOpen,
		stErrGripNotClose,
		stErrInsertNotDown,
		stErrInsertNotUp,
		stErrDriveErr,
		stErrDriveTimeOut,
		stErrDriveHome,
		stErrInitSensor,
		stErrNestSensor

)DINT;
END_TYPE

// ---- DUTs/Stations/machine/machineDisplayStates.TcDUT
{attribute 'qualified_only'}

TYPE machineDisplayStates :
(
	dStStartUp             := 10,
	dStEMGButtonDown,
	dStOpenDoors,
	dStNoAirSupplay,
	dStStationError,
	dStMachineIsStopping,
	dStMachineIsStopped,
	dStAutoRun,
	dStMachineStandBy,
	dStMachinePurgeActive,
	dStMachineRobotEMG,
	dStMachineRobotNoCom
	
)DINT;
END_TYPE

// ---- DUTs/Stations/machine/machineImage.TcDUT
TYPE machineImage :
STRUCT
	
   xDoors 	        	: imageIO := ( stIO   := Stations.machineHmiIO.x_DoorsOK,
									   image  := ADR(Global.INPUT_IMAGE),
									   iType  := ioType.INPUT_BIT,
									   iByte  := 2,
									   iBit   := 5 );	
									   
   xEmgBnt				: imageIO := ( stIO   := Stations.machineHmiIO.x_EmgOK,
									   image  := ADR(Global.INPUT_IMAGE),
									   iType  := ioType.INPUT_BIT,
									   iByte  := 2,
									   iBit   := 4 );

    xAirOk 				: imageIO := ( stIO   := Stations.machineHmiIO.x_AirOk,
									   image  := ADR(Global.INPUT_IMAGE),
									   iType  := ioType.INPUT_BIT,
									   iByte  := 2,
									   iBit   := 0 );
									   
    xRobotEmgOk 		: imageIO := ( stIO   := Stations.machineHmiIO.x_robotEmgOk,
									   image  := ADR(Global.INPUT_IMAGE),
									   iType  := ioType.INPUT_BIT,
									   iByte  := 2,
									   iBit   := 2 );									   
									   									   
    yZumer 				: imageIO := ( stIO   := Stations.machineHmiIO.y_Zumer,
									   image  := ADR(Global.OUTPUT_IMAGE),
									   iType  := ioType.OUTPUT_BIT,
									   iByte  := 6,
									   iBit   := 2 ); 	

	
  
END_STRUCT
END_TYPE

// ---- DUTs/Stations/machine/machineIO.TcDUT
TYPE machineIO :
STRUCT
	
	// Входове
	x_DoorsOK		: BOOL;					    // Вратите са затворени 
	x_EmgOK			: BOOL;					    // Систама за безопасност е активна
	x_AirOk 		: BOOL;						// Има налягане на въздуха
	x_robotEmgOk    : BOOL;
	
	// Изходи
	y_Zumer		    : BOOL;                     // Звуков сигнал
	


END_STRUCT
END_TYPE

// ---- DUTs/Stations/machine/machineSettings.TcDUT
TYPE machineSettings :
STRUCT
END_STRUCT
END_TYPE

// ---- DUTs/Stations/machine/machineStates.TcDUT
{attribute 'qualified_only'}

TYPE machineStates :
(
		stNull      :=    Consts.ST_NULL,
		stStartUp   :=    Consts.ST_START_UP,
		stInit      :=    Consts.ST_INIT,
		stReady     :=    Consts.ST_READY,
		stStop      :=    Consts.ST_STOP,
		stStepBlock :=    Consts.ST_STEP_BLOCK,	
		stEMG		:=    Consts.ST_EMG,
		
		stSafetyStop    :=    1000,
		stCheckState,
		stStopMach,
		stStopping,
		stAutoRun,
		stMachError,
		
	    stPurgeStart,
		stPurgeDialIndexSync,
		stPurgeRobot,
		stPurgeStackers,
		stPurgeDone

)DINT;
END_TYPE

// ---- DUTs/Stations/roboArm/roboArmDisplayStates.TcDUT
{attribute 'qualified_only'}

TYPE roboArmDisplayStates :
(

	dStPowerUp                 := 10,
	dStWaitForNextStep,
	dStWorking,
	
	dStErrGripNotOpen,
	dStErrGripNotClose,
	dStErrSlideNotDown,
	dStErrSlideNotUp,
	dStErrRotatorNotTurn180,
	dStErrRotatorNotTurn0,
	dStErrInitPalletOnWaitPos24,
	dStErrInitPalletOnWaitPos27,
	dStErrInitSensorInGrip,
	dStErrRobotHomeMoveIsTooLong,
	dStErrRobotMoveIsTooLong,
	dStErrRobotError,
	dStErrRobotRecipeLoadIsTooLong,
	dStErrRobotWaitPosIsEmpty,
	dStErrRobotWaitPosIsNotEmpty,
	dStErrRobotNoPalletAtUnloadStacker


)DINT;
END_TYPE

// ---- DUTs/Stations/roboArm/roboArmImage.TcDUT
TYPE roboArmImage :
STRUCT
	
    xGrip_open 	    	: imageIO := ( stIO   := Stations.roboHmiIO.x_Grip_open,
									   image  := ADR(Global.INPUT_IMAGE),
									   iType  := ioType.INPUT_BIT,
									   iByte  := 9,
									   iBit   := 2 );	
									   
    xGrip_close 		: imageIO := ( stIO   := Stations.roboHmiIO.x_Grip_close,
									   image  := ADR(Global.INPUT_IMAGE),
									   iType  := ioType.INPUT_BIT,
									   iByte  := 9,
									   iBit   := 3 );

    xRot_home 	    	: imageIO := ( stIO   := Stations.roboHmiIO.x_Rot_home,
									   image  := ADR(Global.INPUT_IMAGE),
									   iType  := ioType.INPUT_BIT,
									   iByte  := 9,
									   iBit   := 0 );

    xRot_back 		    : imageIO := ( stIO   := Stations.roboHmiIO.x_Rot_back,
									   image  := ADR(Global.INPUT_IMAGE),
									   iType  := ioType.INPUT_BIT,
									   iByte  := 9,
									   iBit   := 1 );	

    xSlide24_up 	   : imageIO := ( stIO   := Stations.roboHmiIO.x_Slide24_up,
									   image  := ADR(Global.INPUT_IMAGE),
									   iType  := ioType.INPUT_BIT,
									   iByte  := 9,
									   iBit   := 4);	

    xSlide24_down 	   : imageIO := ( stIO   := Stations.roboHmiIO.x_Slide24_down,
									   image  := ADR(Global.INPUT_IMAGE),
									   iType  := ioType.INPUT_BIT,
									   iByte  := 9,
									   iBit   := 5);
									   
    xSlide27_up 	   : imageIO := ( stIO   := Stations.roboHmiIO.x_Slide27_up,
									   image  := ADR(Global.INPUT_IMAGE),
									   iType  := ioType.INPUT_BIT,
									   iByte  := 9,
									   iBit   := 6);	

    xSlide27_down 	   : imageIO := ( stIO   := Stations.roboHmiIO.x_Slide27_down,
									   image  := ADR(Global.INPUT_IMAGE),
									   iType  := ioType.INPUT_BIT,
									   iByte  := 9,
									   iBit   := 7);
					   

    xLaser 	           : imageIO := ( stIO   := Stations.roboHmiIO.x_Laser,
									   image  := ADR(Global.INPUT_IMAGE),
									   iType  := ioType.INPUT_BIT,
									   iByte  := 10,
									   iBit   := 0);	

    xWaitPos24 	        : imageIO := ( stIO   := Stations.roboHmiIO.x_waitPos24,
									   image  := ADR(Global.INPUT_IMAGE),
									   iType  := ioType.INPUT_BIT,
									   iByte  := 16,
									   iBit   := 7);

    xWaitPos27 	        : imageIO := ( stIO   := Stations.roboHmiIO.x_waitPos27,
									   image  := ADR(Global.INPUT_IMAGE),
									   iType  := ioType.INPUT_BIT,
									   iByte  := 17,
									   iBit   := 7);								   			   							   
									   
	// Изходи
    yGrip_open 	       : imageIO := ( stIO   := Stations.roboHmiIO.y_Grip_open,
					 				   image  := ADR(Global.OUTPUT_IMAGE),
									   iType  := ioType.OUTPUT_BIT,
									   iByte  := 9,
									   iBit   := 2 );

    yGrip_close 	   : imageIO := ( stIO   := Stations.roboHmiIO.y_Grip_close,
									   image  := ADR(Global.OUTPUT_IMAGE),
									   iType  := ioType.OUTPUT_BIT,
									   iByte  := 9,
									   iBit   := 3 );

    yRot_home 		   : imageIO := ( stIO   := Stations.roboHmiIO.y_Rot_home,
									   image  := ADR(Global.OUTPUT_IMAGE),
									   iType  := ioType.OUTPUT_BIT,
									   iByte  := 9,
									   iBit   := 0 );	

    yRot_back 	       : imageIO := ( stIO   := Stations.roboHmiIO.y_Rot_back,
									   image  := ADR(Global.OUTPUT_IMAGE),
									   iType  := ioType.OUTPUT_BIT,
									   iByte  := 9,
									   iBit   := 1 );	

    ySlide24_up 	       : imageIO := ( stIO   := Stations.roboHmiIO.y_Slide24_up,
									   image  := ADR(Global.OUTPUT_IMAGE),
									   iType  := ioType.OUTPUT_BIT,
									   iByte  := 9,
									   iBit   := 4 );

    ySlide24_down 	   : imageIO := ( stIO   := Stations.roboHmiIO.y_Slide24_down,
									   image  := ADR(Global.OUTPUT_IMAGE),
									   iType  := ioType.OUTPUT_BIT,
									   iByte  := 9,
									   iBit   := 5 );

    yPalletLoad24 	   : imageIO := ( stIO   := Stations.roboHmiIO.y_PalletLoad24,
									   image  := ADR(Global.OUTPUT_IMAGE),
									   iType  := ioType.OUTPUT_BIT,
									   iByte  := 10,
									   iBit   := 0 );		   

    ySlide27_up 	       : imageIO := ( stIO   := Stations.roboHmiIO.y_Slide27_up,
									   image  := ADR(Global.OUTPUT_IMAGE),
									   iType  := ioType.OUTPUT_BIT,
									   iByte  := 9,
									   iBit   := 6 );

    ySlide27_down 	   : imageIO := ( stIO   := Stations.roboHmiIO.y_Slide27_down,
									   image  := ADR(Global.OUTPUT_IMAGE),
									   iType  := ioType.OUTPUT_BIT,
									   iByte  := 9,
									   iBit   := 7 );

    yPalletLoad27 	   : imageIO := ( stIO   := Stations.roboHmiIO.y_PalletLoad27,
									   image  := ADR(Global.OUTPUT_IMAGE),
									   iType  := ioType.OUTPUT_BIT,
									   iByte  := 10,
									   iBit   := 1 );									      
									  						   
    ySignalLamp24 	   : imageIO := ( stIO   := Stations.roboHmiIO.y_signalLamp24,
									   image  := ADR(Global.OUTPUT_IMAGE),
									   iType  := ioType.OUTPUT_BIT,
									   iByte  := 6,
									   iBit   := 0 );	

    ySignalLamp27	   : imageIO := ( stIO   := Stations.roboHmiIO.y_signalLamp27,
									   image  := ADR(Global.OUTPUT_IMAGE),
									   iType  := ioType.OUTPUT_BIT,
									   iByte  := 6,
									   iBit   := 1 );								   
				   	

END_STRUCT
END_TYPE

// ---- DUTs/Stations/roboArm/roboArmIO.TcDUT
TYPE roboArmIO :
STRUCT
	
	// Входове
	x_Grip_open				: BOOL;        //  Грипера на робота е отворен
	x_Grip_close			: BOOL;        //  Грипера на робота е затворен
	x_Rot_home				: BOOL;        //  Ротатора е в home (прав)
	x_Rot_back				: BOOL;        //  Ротатора е завъртян (обърнал е сензор на 180 град.)
	x_Slide24_up			: BOOL;        //  Грипера за тара е свален
	x_Slide24_down          : BOOL;        //  Грипера за тара е вдигнат
	x_Slide27_up			: BOOL;        //  Грипера за тара е свален
	x_Slide27_down          : BOOL;        //  Грипера за тара е вдигнат	
	x_Laser                 : BOOL;        //  Сигнал от лазерната ролетка
	x_waitPos24             : BOOL;        //  Сензор на чакаща поз. HEX24
	x_waitPos27             : BOOL;        //  Сензор на чакаща поз. HEX27
	
	// Изходи
	y_Grip_open				: BOOL;        //  
	y_Grip_close			: BOOL;        //  
	y_Rot_home				: BOOL;        //  
	y_Rot_back				: BOOL;        //  
	y_Slide24_up			: BOOL;        //  
	y_Slide24_down          : BOOL;        // 
	y_Slide27_up			: BOOL;        //  
	y_Slide27_down          : BOOL;        // 
	y_PalletLoad24          : BOOL;        //  Сигнал за захващане/пускане на тара
	y_PalletLoad27          : BOOL;        //  Сигнал за захващане/пускане на тара	
	y_signalLamp24          : BOOL;        //  Сигнална лампа за чакаща поз. HEX24
	y_signalLamp27          : BOOL;        //  Сигнална лампа за чакаща поз. HEX27	
	

END_STRUCT
END_TYPE

// ---- DUTs/Stations/roboArm/roboArmSettings.TcDUT
TYPE roboArmSettings :
STRUCT  PERSISTENT
	
	roboArmParams         : ARRAY[1..Consts.MAX_RECIPE] OF RoboArmsRecipe;


END_STRUCT
END_TYPE

// ---- DUTs/Stations/roboArm/roboArmsRecipe.TcDUT
TYPE roboArmsRecipe :
STRUCT
	
	fixtureNum     : INT    := 48;                    // Брой сензори в тара
	waitPos24      : BOOL   := FALSE;                 // Чакащата позиция е HEX24
	waitPos27      : BOOL   := TRUE;                  // Чакащата позиция е HEX27

END_STRUCT
END_TYPE

// ---- DUTs/Stations/roboArm/roboArmStates.TcDUT
{attribute 'qualified_only'}

TYPE roboArmStates :
(
		stNull      :=    Consts.ST_NULL,
		stStartUp   :=    Consts.ST_START_UP,
		stInit      :=    Consts.ST_INIT,
		stReady     :=    Consts.ST_READY,
		stStop      :=    Consts.ST_STOP,
		stStepBlock :=    Consts.ST_STEP_BLOCK,	
		stEMG		:=    Consts.ST_EMG,
		
		
		
		stPowerUp    :=    1000,
		stInitDone,
		stRobotReset,
		stRobotResetDone,
		stStationStop,
		stNextRobotState,
		
		stPurgeStart,
		stPurgeMove,
		stPurgeMoveCheck,
		stPurgeSync,
		stPurgeMoveDone,
		
		stInitStart,
		stInitMoveHome,
		stInitMoveCheck,
		stInitToolCheck,
		stInitLoadRecipe,
		stInitRecipeCheck,
		stInitSyncStations,
		stInitWaitLoadStacker,
		stInitReady,
		
		stResetStart, 
		stResetSlider,
		stResetSliderCheck,
		stResetGrip,
		stResetGripCheck,
		stResetMoveCheck,
		stResetRotCheck,
		stResetSync,
		stResetDone, 
		
		stMoveToEmptyStart,
		stMoveToEmptyCheck,
		stMoveToEmptyMoveCheck,
		stMoveToEmptySliderDown,
		stMoveToEmptySliderCheck,
		stMoveToEmptyDone,
		
		stEmptyToUnloadStart,
		stEmptyToPalletHome,
		stMoveToUnloadSync, 
		stEmptyToUnloadMove,
		stEmptyToUnloadMoveCheck, 
		stEmptyToUnloadDone,
		
		stUnloadPalletStart,
		stUnloadPalletSyncStacker,
		stUnlodPalletRelease, 
		stUnloadPalletSlideCheck,
		stUnloadPalletSync,
		stUnloadPalletDone,
		
		stLoadPalletStart, 
		stLoadPalletSlideDown,
		stLoadPalletSliderCheck,
		stLoadPalletSignal,
		stLoadPalletSync,
		stLoadPalletDone,
		
		stEmptyPosStart, 
		stEmptyPosPalletHome, 
		stEmptyPosPalletCheck, 
		stEmptyPosMove,
		stEmptyPosMoveCheck,
		stEmptyPosRelease,
		stEmptyPosSlideCheck,
		stEmptyPosSync,
		stEmptyPosDone,
		
		stLoadStart, 
		stLoadMove1,
		stLoadMoveCheck1,
		stLoadWaitCommand,
		stLoadMove2,
		stLoadMoveCheck2,
		stLoadGripCheck,
		stLoadDone,
		
		stUnloadStart, 
		stUnloadMove1,
		stUnloadMoveCheck1,
		stUnloadRotCheck,
		stUnloadMoveCheck2,
		stUnloadGripCheck,
		stUnloadDone, 
		
		stLInsertStart,
		stLInsertMove1,
		stLInsertMoveCheck1,
		stLInsertRotCheck,
		stLInsertMoveCheck2,
		stLInsertMoveDone,
		
		stLInsertLockStart,
		stLInsertLockSync,
		stLInsertLockGripOpen,
		stLInsertLockGripCheck,
		stLInsertLockDone,
		
		stLInsertBackStart,
		stLInsertBackMove,
		stLInsertBackMoveCheck,
		stLInsertBackDone,
		
		stUInsertStart, 
		stUInsertMove1,
		stUInsertMoveCheck1,
		stUInsertRotCheck,
		stUInsertSync,
		stUInsertMove2,
		stUInsertMoveCheck2,
		stUInsertMoveDone,
		
		stUInsertLockStart,
		stUInsertLockGripClose,
		stUInsertLockGripCheck,
		stUInsertLockSync,
		stUInsertLockDone,	
			
        stUInsertBackStart, 
		stUInsertBackMove,
		stUInsertBackMoveCheck,
		stUInsertBackSync,
		stUInsertBackDone,		
		
		stNextMoveStart, 
		stNextMoveWaitLStacker,
		stNextMovePalletCheck,
		stNextMoveSync,
		stNextMovePalletHome, //
		
		stNextMoveCheck1,
		stNextMovePass,
		stNextMoveUnlodeFull,
		stNextMoveEmptyCheck,
		stNextMovePalletOnUload,
		stNextMoveLoadMove,
		stNextMoveLoadMoveCheck,
		stNextMoveLoadDone,
		stNextMoveLoadEmpty,
		stNextMoveCheck2,
		stNextNewCycle,	
		
		stErrGripNotOpen,
		stErrGripNotClose,
		stErrRotNotTurn180,
		stErrRotNotTurn0,
		stErrSlliderNotDown,
		stErrSlideNotUp,
		stErrInitSensor,
		stErrInitPalletOn24,
		stErrInitPalletOn27,
		
		stErrRobot,
		stErrRobotReset,
		stErrRobotTimeOut,
		stErrRobotRecipeTimeOut,
		stErrNoPalletWaitPos,
		stErrPalletOnWaitPos,
		stErrNoPalletUnload,
		stErrRobotCom

)DINT;
END_TYPE

// ---- DUTs/Stations/stackerLoad/palletParamsL.TcDUT
TYPE palletParamsL :
STRUCT
	

	zeroPos                  : REAL;
	size                     : REAL;


END_STRUCT
END_TYPE

// ---- DUTs/Stations/stackerLoad/stackerLoadDisplayStates.TcDUT
{attribute 'qualified_only'}

TYPE stackerLoadDisplayStates :
(
	dStStartingUp 			:= 1000,
	dStStandBy,
	dStStackerIsReseting,
	dStAxisNotConfigured,
	dStRemotePalletManually,
	dStFixerCylinderDidNotOpen,
	dStFixerCylinderDidNotClose,
	dStLock1CylinderDidNotOpen,
	dStLock1CylinderDidNotClose,
	dStLock2CylinderDidNotOpen,
	dStLock2CylinderDidNotClose,
	dStFestoDriveError,
	dStAxisInitMoveTakesTooLong,
	dStWaitForPalletsLoading, 
	dStLoadPallets, 
	dStPalletLoadMoveTakesTooLong,
	dStWaitForPallet,
	dStPalletMoveTakesTooLong,
	dStReleaseEmptyPallet,
    dStThereIsNoPalletOnTop,
	dStStationIsStopped,
	dStWaitForNextStep

	
)DINT;
END_TYPE

// ---- DUTs/Stations/stackerLoad/stackerLoadImage.TcDUT
TYPE stackerLoadImage :
STRUCT
	
  xLock1_lock 	        	   : imageIO := ( stIO  := Stations.sLoadHmiIO.x_Lock1_lock,
									   image  		  := ADR(Global.INPUT_IMAGE),
									   iType  		  := ioType.INPUT_BIT,
									   iByte 		  := 16,
									   iBit  		  := 0 );	
									   
   xLock1_unlock				: imageIO := ( stIO   := Stations.sLoadHmiIO.x_Lock1_unlock,
									   image 		  := ADR(Global.INPUT_IMAGE),
									   iType  		  := ioType.INPUT_BIT,
									   iByte 		  := 16,
									   iBit   		  := 1 );

    xLock2_lock 				: imageIO := ( stIO   := Stations.sLoadHmiIO.x_Lock2_lock,
									   image  		  := ADR(Global.INPUT_IMAGE),
									   iType  		  := ioType.INPUT_BIT,
									   iByte 		  := 16,
									   iBit   		  := 2 );
									  
    xLock2_unlock 				: imageIO := ( stIO   := Stations.sLoadHmiIO.x_Lock2_unlock,
									   image  		  := ADR(Global.INPUT_IMAGE),
									   iType  		  := ioType.INPUT_BIT,
									   iByte 		  := 16,
									   iBit   		  := 3 );

    xPalletOnTop27 				: imageIO := ( stIO   := Stations.sLoadHmiIO.x_PalletOnTop27,
									   image  		  := ADR(Global.INPUT_IMAGE),
									   iType  		  := ioType.INPUT_BIT,
									   iByte 		  := 16,
									   iBit   		  := 6 );
									   
	xPalletOnTop24 				: imageIO := ( stIO   := Stations.sLoadHmiIO.x_PalletOnTop24,
									   image  		  := ADR(Global.INPUT_IMAGE),
									   iType  		  := ioType.INPUT_BIT,
									   iByte 		  := 3,
									   iBit   		  := 2 );								   

    xPalletFix_lock 				: imageIO := ( stIO   := Stations.sLoadHmiIO.x_PalletFix_lock,
									   image  		  := ADR(Global.INPUT_IMAGE),
									   iType  		  := ioType.INPUT_BIT,
									   iByte 		  := 16,
									   iBit   		  := 5 );

    xPalletFix_unlock 				: imageIO := ( stIO   := Stations.sLoadHmiIO.x_PalletFix_unlock,
									   image  		  := ADR(Global.INPUT_IMAGE),
									   iType  		  := ioType.INPUT_BIT,
									   iByte 		  := 16,
									   iBit   		  := 4 );

    yLock1_lock 				: imageIO := ( stIO   := Stations.sLoadHmiIO.y_Lock1_lock,
									   image  		  := ADR(Global.OUTPUT_IMAGE),
									   iType  		  := ioType.OUTPUT_BIT,
									   iByte 		  := 151,
									   iBit   		  := 1 ); 

    yLock1_unlock 				: imageIO := ( stIO   := Stations.sLoadHmiIO.y_Lock1_unlock,
									   image  		  := ADR(Global.OUTPUT_IMAGE),
									   iType  		  := ioType.OUTPUT_BIT,
									   iByte 		  := 151,
									   iBit   		  := 0 ); 
									   

    yLock2_lock 				: imageIO := ( stIO   := Stations.sLoadHmiIO.y_Lock2_lock,
									   image  		  := ADR(Global.OUTPUT_IMAGE),
									   iType  		  := ioType.OUTPUT_BIT,
									   iByte 		  := 152,
									   iBit   		  := 0 ); 

    yLock2_unlock 				: imageIO := ( stIO   := Stations.sLoadHmiIO.y_Lock2_unlock,
									   image  		  := ADR(Global.OUTPUT_IMAGE),
									   iType  		  := ioType.OUTPUT_BIT,
									   iByte 		  := 152,
									   iBit   		  := 1 );									   

 
    yPalletFix_lock 				: imageIO := ( stIO   := Stations.sLoadHmiIO.y_PalletFix_lock,
									   image  		  := ADR(Global.OUTPUT_IMAGE),
									   iType  		  := ioType.OUTPUT_BIT,
									   iByte 		  := 151,
									   iBit   		  := 5 ); 
									   
    yPalletFix_unlock 				: imageIO := ( stIO   := Stations.sLoadHmiIO.y_PalletFix_unlock,
									   image  		  := ADR(Global.OUTPUT_IMAGE),
									   iType  		  := ioType.OUTPUT_BIT,
									   iByte 		  := 151,
									   iBit   		  := 4 ); 							    

END_STRUCT
END_TYPE

// ---- DUTs/Stations/stackerLoad/stackerLoadIO.TcDUT
TYPE stackerLoadIO :
STRUCT
	
	// Входове
	x_Lock1_lock				: BOOL;        // Сензор цилиндър на заключалка 1 на тара - тарата е ЗАКЛЮЧЕНА
	x_Lock1_unlock				: BOOL;        // Сензор цилиндър на заключалка 1 на тара - тарата е ОТКЛЮЧЕНА
	x_Lock2_lock				: BOOL;        // Сензор цилиндър на заключалка 2 на тара - тарата е ЗАКЛЮЧЕНА
	x_Lock2_unlock				: BOOL;        // Сензор цилиндър на заключалка 2 на тара - тарата е ОТКЛЮЧЕНА
	x_PalletOnTop27				: BOOL;        // Дифузен сензор на върха на стакера - ИМА тара за заключване
	x_PalletOnTop24				: BOOL;        // Дифузен сензор на върха на стакера - ИМА тара за заключване
	x_PalletFix_lock			: BOOL; 	   // Сензор цилиндър за фиксиране на тарата - тарата е ЗАКЛЮЧЕНА
	x_PalletFix_unlock			: BOOL; 	   // Сензор цилиндър за фиксиране на тарата - тарата e ОТКЛЮЧЕНА
	
	// Изходи
	y_Lock1_lock				: BOOL;        // Пневно сигнал на заключалка 1 на тара - ЗАКЛЮЧВАНЕ
	y_Lock1_unlock				: BOOL;        // Пневно сигнал на заключалка 1 на тара - ОТКЛЮЧВАНЕ
	y_Lock2_lock				: BOOL;        // Пневно сигнал на заключалка 1 на тара - ЗАКЛЮЧВАНЕ
	y_Lock2_unlock				: BOOL;        // Пневно сигнал на заключалка 1 на тара - ОТКЛЮЧВАНЕ
	y_PalletFix_lock            : BOOL; 	   // Пневно сигнал за фиксиране на тара - ЗАКЛЮЧВАНЕ
    y_PalletFix_unlock          : BOOL; 	   // Пневно сигнал за фиксиране на тара - ОТКЛЮЧЕНА


	
END_STRUCT
END_TYPE

// ---- DUTs/Stations/stackerLoad/stackerLoadSettings.TcDUT
TYPE stackerLoadSettings :
STRUCT
	
	axisLength                :   REAL   := 625; 		   // макс ход на оста на стакера за модел HEX 24
	axisWorkSpeed             :	  REAL   := 200; 	       // скорост 
	axisInitSpeed			  :   REAL   := 200; 	       // скорост при движение нагоре (при init)
	axisAcc					  :   REAL   := 200 ;          // ускр.
	pallet                    :   ARRAY[1..Consts.MAX_RECIPE] OF palletParamsL; 

END_STRUCT
END_TYPE

// ---- DUTs/Stations/stackerLoad/stackerLoadStates.TcDUT
{attribute 'qualified_only'}

TYPE stackerLoadStates :
(
		stNull      :=    Consts.ST_NULL,
		stStartUp   :=    Consts.ST_START_UP,
		stInit      :=    Consts.ST_INIT,
		stReady     :=    Consts.ST_READY,
		stStop      :=    Consts.ST_STOP,
		stStepBlock :=    Consts.ST_STEP_BLOCK,	
		stEMG		:=    Consts.ST_EMG,
		 
		stPowerUp    :=    1000,
		stStackerStopped,
		stInitDone,
		
		stResetStart,
		stResetCheckLocks,
		stResetUnlockPallet,
		stResetEnableDrive,
		stResetDriveMove,
		stResetCheckDrive,
		stResetDone,
		
		stLoadPalletsStart, 
		stPalletsLoadLimitCheck,
		stPalletsLoadCalcAxis,
		stPalletsLoadCheckTop,
		stPalletsLoadCheckLocks,
		stLoadPalletsDriveOn,
		stLoadPalletsCalcPos,
		stLoadPalletsMoveDone,
		stLoadPalletsMoveAgain,
		stLoadPalletsDone, 
		
		stPreparePalletStart,
		stPreparePalletCheckTop,
		stPreparePalletCheckLocks1,
		stPreparePalletSyncRobot,
		stPrepareDriveOn,
		stPreparePalletMove,
		stPreparePalletMoveCheck,
		stPreparePalletLock,
		stPreparePalletDone,
		
		stMoveDownStart,
		stMoveDownCkeckTop,
		stMoveDownCheckLocks,
		stMoveDownCheckFix, 
		stMoveSync,
		stMoveDownDriveOn,
		stMoveDownMove,
		stMoveDownMoveCheck,
		stMoveDownDone,
		
		stReleasePalletStart, 
		stReleasePalletUnlock,
		stReleasePalletUnlockCheck,
		stReleasePalletSignalRobot,
		stReleasePalletDone, 
		
		stRoboOutStart,
		stRoboOutDone,
		
		stLoadPurgeStart,
		stLoadPurgeCheck,
		stLoadPurgeDriveOn,
		stLoadPurgeMove,
		stLoadPurgeMoveCheck,
		stLoadPurgeDone,
		stLoadPurgeConfirm,
		
		
		stErrNoProperSettings,
		stErrRemovePallet,
		stErrFixerNotOpen,
		stErrFixerNotClose,
		stErrLock1NotClose,
		stErrLock1NotOpen,
		stErrLock2NotClose,
		stErrLock2NotOpen,
		stErrAxis,
		stInitMoveErr,
		stErrPalletLoad,
		stErrPalletMove,
		stErrNoPallet


)DINT;
END_TYPE

// ---- DUTs/stationBase.TcDUT
TYPE stationBase :
STRUCT
	
	StationID						: DINT;
	StationType						: DINT;
	Ready							: BOOL;
	Busy							: BOOL;
	Error							: BOOL;
	Disabled						: BOOL;
	CurrentState					: DINT;
	LastState						: DINT;
	LastErrorState					: DINT;
	DisplayState					: DINT;
	DependencyState					: DINT;	     
	DoInit							: BOOL;       // това е бутона RESET на HMI - да се добави
	DoStart							: BOOL;       // след като е бил в StepMode с този бутон продължава на AutoMode
	DoEnd							: BOOL;       // не се ползва - да не се добавя бутона на HMI
	DoStop							: BOOL;
	DoRetry							: BOOL;       // не се ползва - да не се добавя бутона на HMI
	DoConfirmDependency				: BOOL;       
	ToggleEnable					: BOOL;
	AutoMode						: BOOL;
	NextStep						: BOOL;
	
END_STRUCT
END_TYPE

// ---- DUTs/Stations/stackerUnload/palletParamsU.TcDUT
TYPE palletParamsU :
STRUCT
	
	zeroPos             : REAL;
    moveDownStep		: REAL;
	moveUpStep 			: REAL;



END_STRUCT
END_TYPE

// ---- DUTs/Stations/stackerUnload/stackerUnLoadDisplayStates.TcDUT
{attribute 'qualified_only'}

TYPE stackerUnLoadDisplayStates :
(
	dStStartingUp 			:= 1000,
	dStStandBy,
	dStStackerIsReseting,
	dStPalletReady,
    dStAxisNotConfigured,	
	dStRemotePalletManually,
	dStLock1CylinderDidNotOpen,
    dStLock1CylinderDidNotClose,
	dStLock2CylinderDidNotOpen,
	dStLock2CylinderDidNotClose,
    dStFixerCylinderDidNotOpen,	
    dStFixerCylinderDidNotClose,
    dStFestoDriveError,	
    dStAxisInitMoveTakesTooLong,	
	dStPalletMoveTakesTooLong,
    dStPalletIsDetectedFault,
    dStThereIsNoPalletOnTop,	
	dStWaitForNextStep,
	dStStationIsStopped
	
	
)DINT;
END_TYPE

// ---- DUTs/Stations/stackerUnload/stackerUnLoadImage.TcDUT
TYPE stackerUnLoadImage :
STRUCT
	xLock1_lock 	        	   : imageIO := ( stIO  := Stations.sUnloadHmiIO.x_Lock1_lock,
									   image  		:= ADR(Global.INPUT_IMAGE),
									   iType  		:= ioType.INPUT_BIT,
									   iByte 		:= 17,
									   iBit  		:= 0 );	
									   
   xLock1_unlock				: imageIO := ( stIO   := Stations.sUnloadHmiIO.x_Lock1_unlock,
									   image 		  := ADR(Global.INPUT_IMAGE),
									   iType  		  := ioType.INPUT_BIT,
									   iByte 		  := 17,
									   iBit   		  := 1 );

    xLock2_lock 				: imageIO := ( stIO   := Stations.sUnloadHmiIO.x_Lock2_lock,
									   image  		  := ADR(Global.INPUT_IMAGE),
									   iType  		  := ioType.INPUT_BIT,
									   iByte 		  := 17,
									   iBit   		  := 2 );
									  
    xLock2_unlock 				: imageIO := ( stIO   := Stations.sUnloadHmiIO.x_Lock2_unlock,
									   image  		  := ADR(Global.INPUT_IMAGE),
									   iType  		  := ioType.INPUT_BIT,
									   iByte 		  := 17,
									   iBit   		  := 3 );

    xPalletOnTop 				: imageIO := ( stIO   := Stations.sUnloadHmiIO.x_PalletOnTop,
									   image  		  := ADR(Global.INPUT_IMAGE),
									   iType  		  := ioType.INPUT_BIT,
									   iByte 		  := 17,
									   iBit   		  := 6 );

    xPalletFix_lock 				: imageIO := ( stIO   := Stations.sUnloadHmiIO.x_PalletFix_lock,
									   image  		  := ADR(Global.INPUT_IMAGE),
									   iType  		  := ioType.INPUT_BIT,
									   iByte 		  := 17,
									   iBit   		  := 4 );

    xPalletFix_unlock 				: imageIO := ( stIO   := Stations.sUnloadHmiIO.x_PalletFix_unlock,
									   image  		  := ADR(Global.INPUT_IMAGE),
									   iType  		  := ioType.INPUT_BIT,
									   iByte 		  := 17,
									   iBit   		  := 5 );

    yLock1_lock 				: imageIO := ( stIO   := Stations.sUnloadHmiIO.y_Lock1_lock,
									   image  		  := ADR(Global.OUTPUT_IMAGE),
									   iType  		  := ioType.OUTPUT_BIT,
									   iByte 		  := 151,
									   iBit   		  := 3 ); 

    yLock1_unlock 				: imageIO := ( stIO   := Stations.sUnloadHmiIO.y_Lock1_unlock,
									   image  		  := ADR(Global.OUTPUT_IMAGE),
									   iType  		  := ioType.OUTPUT_BIT,
									   iByte 		  := 151,
									   iBit   		  := 2 ); 
									   
    yLock2_lock 				: imageIO := ( stIO   := Stations.sUnloadHmiIO.y_Lock2_lock,
									   image  		  := ADR(Global.OUTPUT_IMAGE),
									   iType  		  := ioType.OUTPUT_BIT,
									   iByte 		  := 151,
									   iBit   		  := 3 ); 

    yLock2_unlock 				: imageIO := ( stIO   := Stations.sUnloadHmiIO.y_Lock2_unlock,
									   image  		  := ADR(Global.OUTPUT_IMAGE),
									   iType  		  := ioType.OUTPUT_BIT,
									   iByte 		  := 151,
									   iBit   		  := 2 ); 									   
 
    yPalletFix_lock 				: imageIO := ( stIO   := Stations.sUnloadHmiIO.y_PalletFix_lock,
									   image  		  := ADR(Global.OUTPUT_IMAGE),
									   iType  		  := ioType.OUTPUT_BIT,
									   iByte 		  := 151,
									   iBit   		  := 6 ); 
									   
    yPalletFix_unlock 				: imageIO := ( stIO   := Stations.sUnloadHmiIO.y_PalletFix_unlock,
									   image  		  := ADR(Global.OUTPUT_IMAGE),
									   iType  		  := ioType.OUTPUT_BIT,
									   iByte 		  := 151,
									   iBit   		  := 7 ); 
								
END_STRUCT
END_TYPE

// ---- DUTs/Stations/stackerUnload/stackerUnLoadIO.TcDUT
TYPE stackerUnLoadIO :
STRUCT
	
	// Входове
	x_Lock1_lock				: BOOL;        // Сензор цилиндър на заключалка 1 на тара - тарата е ЗАКЛЮЧЕНА
	x_Lock1_unlock				: BOOL;        // Сензор цилиндър на заключалка 1 на тара - тарата е ОТКЛЮЧЕНА
	x_Lock2_lock				: BOOL;        // Сензор цилиндър на заключалка 2 на тара - тарата е ЗАКЛЮЧЕНА
	x_Lock2_unlock				: BOOL;        // Сензор цилиндър на заключалка 2 на тара - тарата е ОТКЛЮЧЕНА
	x_PalletOnTop				: BOOL;        // Дифузен сензор на върха на стакера - ИМА тара за заключване
	x_PalletFix_lock			: BOOL; 	   // Сензор цилиндър за фиксиране на тарата - тарата е ЗАКЛЮЧЕНА
	x_PalletFix_unlock			: BOOL; 	   // Сензор цилиндър за фиксиране на тарата - тарата e ОТКЛЮЧЕНА
	
	// Изходи
	y_Lock1_lock				: BOOL;        // Пневно сигнал на заключалка 1 на тара - ЗАКЛЮЧВАНЕ
	y_Lock1_unlock				: BOOL;        // Пневно сигнал на заключалка 1 на тара - ОТКЛЮЧВАНЕ
	y_Lock2_lock				: BOOL;        // Пневно сигнал на заключалка 2 на тара - ЗАКЛЮЧВАНЕ
	y_Lock2_unlock				: BOOL;        // Пневно сигнал на заключалка 2 на тара - ОТКЛЮЧВАНЕ	
	y_PalletFix_lock            : BOOL; 	   // Пневно сигнал за фиксиране на тара - ЗАКЛЮЧВАНЕ
    y_PalletFix_unlock          : BOOL; 	   // Пневно сигнал за фиксиране на тара - ОТКЛЮЧЕНА

END_STRUCT
END_TYPE

// ---- DUTs/Stations/stackerUnload/stackerUnLoadSettings.TcDUT
TYPE stackerUnLoadSettings :
STRUCT
	
	axisLength                :   REAL   := 625.0; 		    // макс ход на оста на стакера за модел HEX 24
	axisWorkSpeed             :	  REAL   := 200.0; 	        // скорост 
	axisInitSpeed			  :   REAL   := 200.0; 	        // скорост при движение нагоре (при init)
	axisAcc					  :   REAL   := 200.0 ;         // ускр.
	pallet                    :   ARRAY[1..Consts.MAX_RECIPE] OF palletParamsU; 

END_STRUCT
END_TYPE

// ---- DUTs/Stations/stackerUnload/stackerUnLoadStates.TcDUT
{attribute 'qualified_only'}

TYPE stackerUnLoadStates :
(
		stNull      :=    Consts.ST_NULL,
		stStartUp   :=    Consts.ST_START_UP,
		stInit      :=    Consts.ST_INIT,
		stReady     :=    Consts.ST_READY,
		stStop      :=    Consts.ST_STOP,
		stStepBlock :=    Consts.ST_STEP_BLOCK,	
		stEMG		:=    Consts.ST_EMG,
		 
		stPowerUp    :=    1000,
		stStackerStopped,
		stInitDone,
		
		stResetStart,
		stResetOpenLocks,
		stResetCheckLocks,
		stResetEnableDrive,
		stResetDriveMove,
		stResetCheckDrive,
		stResetDone,
		
		stPrepareStart,
		stPreparaCheckTop,
		stPrepareLimitCheck,
		stPrepareCalcAxis,
		stPrepareOpenLocks,
		stPrepareCheckLocks,
		stPrepareDriveOn,
		stPrepareDriveMove,
		stPrepareCheckDrive,
		stPrepareSync,
		stPrepareDone,
		
		stMoveUpStart,
		stMoveUpDriveOn,
		stMoveUpDriveMove,
		stMoveUpCkeckDrive,
		stMoveUpDone,
		
		stUnlockPalletStart,
		stUnlockPalletRelease,
		stUnlockPalletCheck,
		stUnlockPalletDriveOn,
		stUnlockPalletDriveMove,
		stUnlockPalletCkeckDrive,   
		stUnlockPalletSync,
		stUnlockPalletDone,
		
		stLockPalletStart,
		stLockPalletLocking,
		stLockPalletCheckLocks,
		stLockPalletSyncRobot,
		stLockPalletLockFix,
		stLockPalletCheckFix,
		stLockPalletDone,
		
		stUnloadPurgeStart,
		stUnloadPurgeCheck,
		stUnloadPurgeDriveOn,
		stUnloadPurgeMove,
		stUnloadPurgeMoveCheck,
		stUnloadPurgeDone,
		stUnloadPurgeConfirm,
		
		
		stErrNoProperSettings,
		stErrRemovePallet,
		stErrFixerNotOpen,
		stErrFixerNotClose,
		stErrLock1NotClose,
		stErrLock1NotOpen,
		stErrLock2NotClose,
		stErrLock2NotOpen,
		stErrAxis,
		stInitMoveErr,
		stErrPalletDetected,
		stErrPalletMove,
		stErrNoPallet

)DINT;
END_TYPE

// ---- POUs/Mitsubishi/DUT/Communication/PacketsStructure/Input/ST_Robot_Mitsubishi_Packet_1000.TcDUT
TYPE ST_Robot_Mitsubishi_Packet_1000 :
STRUCT	
	// Packet number - 1000.
	// From robot.
	// Main robot status packet.
	// Cyclic.
	
	Header							: DINT := 1000;													// Packet header.
	
	Ready							: BIT;															// Is the robot ready for operation.
	Busy							: BIT;															// Is the robot operating.
	Error							: BIT;															// Is the robot in an error state.
	PoweredOn						: BIT;															// Is the robot in a powered on state.
	
	// Not avalable - fillers.
	AutomaticMode					: BIT;
	Executing						: BIT;
	Ending							: BIT;
	ProgramCompleted				: BIT;															// Is the last started program completed.
	GripperA_Present				: BIT;
	GripperB_Present				: BIT;
	GripperA_Open					: BIT;
	GripperB_Open					: BIT;
	NA13							: BIT;
	NA14							: BIT;
	NA15							: BIT;
	NA16							: BIT;
	NA17							: BIT;	
	NA18							: BIT;	
	NA19							: BIT;	
	NA20							: BIT;	
	NA21							: BIT;	
	NA22							: BIT;	
	NA23							: BIT;	
	NA24							: BIT;	
	NA25							: BIT;	
	NA26							: BIT;	
	NA27							: BIT;	
	NA28							: BIT;	
	NA29							: BIT;	
	NA30							: BIT;	
	NA31							: BIT;	
	NA32							: BIT;	
	
	CurrentState					: DINT;															// The current robot state ID if defined.
	CurrentProgram					: DINT;															// The currently selected robot program.
	CurrentTrayPosition				: DINT;															// The currently selected station to work with.
	CurrentSpeed					: DINT;															// The current speed overdive.
	CurrentProductID				: DINT;															// The current product ID if any.
	CurrentGripperID				: DINT;															// The current gripper ID if selected.
	CurrentTrayOrient				: DINT;
	
	CurrentTargetProgram			: DINT;															// The current target robot program.			// | These could be moved in a separate packet.
	CurrentTargetTrayPosition		: DINT;															// The current target robot station.			// |
	CurrentTargetSpeed				: DINT;															// The current target robot speed override.		// |
	CurrentTargetProductID			: DINT;															// The current target product ID.
	CurrentTargetGripperID			: DINT;															// The current target robot gripper ID.		// |
	CurrentTargetTrayOrient			: DINT;															// The current target robot gripper ID.		// 
END_STRUCT
END_TYPE

// ---- POUs/Mitsubishi/DUT/Communication/PacketsStructure/Input/ST_Robot_Mitsubishi_Packet_1100.TcDUT
TYPE ST_Robot_Mitsubishi_Packet_1100 :
STRUCT
	// Packet number - 1100.
	// From robot.
	// Robot base position for station packet.
	// Trigger.
	
	Header							: DINT := 1100;													// Packet header.
	
	CurrentStation					: DINT;															// The currently selected station the robot is working with.
	CorrectionID					: DINT;															// Correction ID.
	
	XValue							: DINT;															// Position X value.
	YValue							: DINT;															// Position Y value.
	ZValue							: DINT;															// Position Z value.
	AValue							: DINT;															// Position A value.
	BValue							: DINT;															// Position B value.
	CValue							: DINT;															// Position C value.
	L1Value							: DINT;															// Position L1 value.
	L2Value							: DINT;															// Position L2 value.
	FLG1Value						: DINT;															// Position FLG1 value.
	FLG2Value						: DINT;															// Position FLG2 value.
END_STRUCT
END_TYPE

// ---- POUs/Mitsubishi/DUT/Communication/PacketsStructure/Input/ST_Robot_Mitsubishi_Packet_1101.TcDUT
TYPE ST_Robot_Mitsubishi_Packet_1101 :
STRUCT
	// Packet number - 1100. 8B This is separated due to the need of on trigger confirmation.
	// From robot.
	// Robot packet received.
	// Trigger.
	
	Header							: DINT := 1101;													// Packet header.
	
	LastReceivedPacketID			: DINT;
END_STRUCT
END_TYPE

// ---- POUs/Mitsubishi/DUT/Communication/PacketsStructure/Input/ST_Robot_Mitsubishi_Packet_1102.TcDUT
TYPE ST_Robot_Mitsubishi_Packet_1102 :
STRUCT
	// Packet number - 1100. 8B This is separated due to the need of on trigger confirmation.
	// From robot.
	// Robot program completed.
	// Trigger.
	
	Header							: DINT := 1102;													// Packet header.
	
	LastProgram						: DINT;
END_STRUCT
END_TYPE

// ---- POUs/Mitsubishi/DUT/Communication/PacketsStructure/Input/ST_Robot_Mitsubishi_Packet_1103.TcDUT
TYPE ST_Robot_Mitsubishi_Packet_1103 :
STRUCT
	// Packet number - 1103. 8B This is separated due to the need of on trigger confirmation.
	// From robot.
	// Robot Dependency confirmed.
	// Trigger.
	
	Header							: DINT := 1103;													// Packet header.
	
	DepencencyState					: DINT;
END_STRUCT
END_TYPE

// ---- POUs/Mitsubishi/DUT/Communication/PacketsStructure/Output/ST_Robot_Mitsubishi_Packet_2000.TcDUT
TYPE ST_Robot_Mitsubishi_Packet_2000 :
STRUCT
	// Packet number - 2000. 48B
	// To robot.
	// Robot Settings packet.
	// Trigger.
	
	Header							: DINT := 2000;													// Packet header.
	
	StartProgram					: BIT;
	// Not avalable - fillers.															// Change the selected station to the target station if possible.
	NA2								: BIT;	
	NA3								: BIT;	
	NA4								: BIT;	
	NA5								: BIT;	
	NA6								: BIT;	
	NA7								: BIT;	
	NA8								: BIT;	
	NA9								: BIT;	
	NA10							: BIT;	
	NA11							: BIT;	
	NA12							: BIT;		
	NA13							: BIT;	
	NA14							: BIT;	
	NA15							: BIT;	
	NA16							: BIT;	
	NA17							: BIT;	
	NA18							: BIT;	
	NA19							: BIT;	
	NA20							: BIT;	
	NA21							: BIT;	
	NA22							: BIT;	
	NA23							: BIT;	
	NA24							: BIT;	
	NA25							: BIT;	
	NA26							: BIT;	
	NA27							: BIT;	
	NA28							: BIT;	
	NA29							: BIT;	
	NA30							: BIT;	
	NA31							: BIT;	
	NA32							: BIT;	
	
	TargetTrayPosition				: DINT;		// The station of interest to be worked with.
	TargetProgram					: DINT;		// The program to be executed.
	TargetSpeed						: DINT;		// The speed overdrive to be set.
	TargetProductID					: DINT;		// Targer Product ID
	TargetGripperID					: DINT;		// Targer Tray Variation
	TargetTrayOrientation			: DINT;		// Targer Tray Orientation
END_STRUCT
END_TYPE

// ---- POUs/Mitsubishi/DUT/Communication/PacketsStructure/Output/ST_Robot_Mitsubishi_Packet_2010.TcDUT
TYPE ST_Robot_Mitsubishi_Packet_2010 :
STRUCT
	// Packet number - 2010.
	// To robot.
	// Robot servo power control packet.
	// Trigger.
	
	Header							: DINT := 2010;	//7DA // Packet header.
	
	Reset 							: BIT; 	//000007DA00000001
	ServoOn							: BIT;	//000007DA00000002
	ServoOff						: BIT;	//000007DA00000004			
	End								: BIT;	//000007DA00000008
	Stop							: BIT;	//000007DA00000010
	Start							: BIT;	//000007DA00000020
		// Not avalable - fillers.
	OpenGripperA					 :BIT;	//000007DA00000040
	CloseGripperA					: BIT;	//000007DA00000080
	OpenGripperB					: BIT;	//000007DA00000100
	CloseGripperB					: BIT;	//000007DA00000200
	NA11							: BIT;	
	NA12							: BIT;
	NA13							: BIT;	
	NA14							: BIT;	
	NA15							: BIT;	
	NA16							: BIT;	
	NA17							: BIT;	
	NA18							: BIT;	
	NA19							: BIT;	
	NA20							: BIT;	
	NA21							: BIT;	
	NA22							: BIT;	
	NA23							: BIT;	
	NA24							: BIT;	
	NA25							: BIT;	
	NA26							: BIT;	
	NA27							: BIT;	
	NA28							: BIT;	
	NA29							: BIT;	
	NA30							: BIT;	
	NA31							: BIT;	
	NA32							: BIT;	
END_STRUCT
END_TYPE

// ---- POUs/Mitsubishi/DUT/Communication/PacketsStructure/Output/ST_Robot_Mitsubishi_Packet_2011.TcDUT
TYPE ST_Robot_Mitsubishi_Packet_2011 :
STRUCT
	// Packet number - 2011.
	// To robot.
	// Robot step control packet.
	// Trigger.
	
	Header							: DINT := 2011;													// Packet header.
	
	StepDirection					: DINT;															// 0 for step Backward, 1 for step Forward.
	
END_STRUCT
END_TYPE

// ---- POUs/Mitsubishi/DUT/Communication/PacketsStructure/Output/ST_Robot_Mitsubishi_Packet_2012.TcDUT
TYPE ST_Robot_Mitsubishi_Packet_2012 :
STRUCT
	// Packet number - 2012.
	// To robot.
	// Robot cycle control packet.
	// Trigger.
	
	Header							: DINT := 2012;													// Packet header.
	
	TargetState						: DINT;															// 0 for cycle End, 1 for cycle Start.
	
END_STRUCT
END_TYPE

// ---- POUs/Mitsubishi/DUT/Communication/PacketsStructure/Output/ST_Robot_Mitsubishi_Packet_2013.TcDUT
TYPE ST_Robot_Mitsubishi_Packet_2013 :
STRUCT
	// Packet number - 2013.
	// To robot.
	// Robot stop control packet.
	// Trigger.
	
	Header							: DINT := 2013;													// Packet header.

END_STRUCT
END_TYPE

// ---- POUs/Mitsubishi/DUT/Communication/PacketsStructure/Output/ST_Robot_Mitsubishi_Packet_2014.TcDUT
TYPE ST_Robot_Mitsubishi_Packet_2014 :
STRUCT
	// Packet number - 2014.
	// To robot.
	// Robot change target station control packet.
	// Trigger.
	
	Header							: DINT := 2014;													// Packet header.
	
	TargetStation					: DINT;															// The station to be switched to.
	
END_STRUCT
END_TYPE

// ---- POUs/Mitsubishi/DUT/Communication/PacketsStructure/Output/ST_Robot_Mitsubishi_Packet_2015.TcDUT
TYPE ST_Robot_Mitsubishi_Packet_2015 :
STRUCT
	// Packet number - 2015.
	// To robot.
	// Robot change target program control packet.
	// Trigger.
	
	Header							: DINT := 2015;													// Packet header.
	
	TargetProgram					: DINT;															// The program to be executed.

END_STRUCT
END_TYPE

// ---- POUs/Mitsubishi/DUT/Communication/PacketsStructure/Output/ST_Robot_Mitsubishi_Packet_2016.TcDUT
TYPE ST_Robot_Mitsubishi_Packet_2016 :
STRUCT
	// Packet number - 2016.
	// To robot.
	// Robot change speed override control packet.
	// Trigger.
	
	Header							: DINT := 2016;													// Packet header.
	
	TargetSpeed						: DINT;															// The speed overdrive to be set.
	
END_STRUCT
END_TYPE

// ---- POUs/Mitsubishi/DUT/Communication/PacketsStructure/Output/ST_Robot_Mitsubishi_Packet_2017.TcDUT
TYPE ST_Robot_Mitsubishi_Packet_2017 :
STRUCT
	// Packet number - 2017.
	// To robot.
	// Robot change target correction id control packet.
	// Trigger.
	
	Header							: DINT := 2017;													// Packet header.
	
	TargetCorrectionID				: DINT;															// The target correction ID.																
	
END_STRUCT
END_TYPE

// ---- POUs/Mitsubishi/DUT/Communication/PacketsStructure/Output/ST_Robot_Mitsubishi_Packet_2018.TcDUT
TYPE ST_Robot_Mitsubishi_Packet_2018 :
STRUCT
	// Packet number - 2018.
	// To robot.
	// Robot dependency state confirmation control packet.
	// Trigger.
	
	Header							: DINT := 2018;													// Packet header.
	
	StateID							: DINT; 														// The state to be confirmed.
	
END_STRUCT
END_TYPE

// ---- POUs/Mitsubishi/DUT/Communication/PacketsStructure/Output/ST_Robot_Mitsubishi_Packet_2019.TcDUT
TYPE ST_Robot_Mitsubishi_Packet_2019 :
STRUCT
	// Packet number - 2019.
	// To robot.
	// Robot start program packet.
	// Trigger.
	
	Header							: DINT := 2019;													// Packet header.
	
	ProgramNumber					: DINT; 														// The program to be started.
	
END_STRUCT
END_TYPE

// ---- POUs/Mitsubishi/DUT/Communication/PacketsStructure/Output/ST_Robot_Mitsubishi_Packet_2100.TcDUT
TYPE ST_Robot_Mitsubishi_Packet_2100 :
STRUCT
	// Packet number - 2100.
	// To robot.
	// Robot correction (data) packet.
	// Trigger.
	
	Header							: DINT := 2100;													// Packet header.
	
	CorrectionID					: DINT;															// Correction ID.
	
	XCorrection						: DINT;															// Position X correction.
	YCorrection						: DINT;															// Position Y correction.
	ZCorrection						: DINT;															// Position Z correction.
	ACorrection						: DINT;															// Position A correction.
	BCorrection						: DINT;															// Position B correction.
	CCorrection						: DINT;															// Position C correction.
	L1Correction					: DINT;															// Position L1 correction.
	L2Correction					: DINT;															// Position L2 correction.
	FLG1Correction					: DINT;															// Position FLG1 correction.
	FLG2Correction					: DINT;															// Position FLG2 correction.
	
END_STRUCT
END_TYPE

// ---- POUs/Mitsubishi/DUT/Communication/PacketsStructure/Output/ST_Robot_Mitsubishi_Packet_2101.TcDUT
TYPE ST_Robot_Mitsubishi_Packet_2101 :
STRUCT
	// Packet number - 2101.
	// To robot.
	// Robot target product ID packet.
	// Trigger.
	
	Header							: DINT := 2101;													// Packet header.
	
	TargetProductID					: DINT;															// The station to be switched to.			// Sumbit as DINT(ROUND(<LREAL>, 2) * 100)
	// TargetProductID					: LREAL;															// The product ID to be switched to.		// On error use top
	
END_STRUCT
END_TYPE

// ---- POUs/Mitsubishi/DUT/Communication/ST_Robot_Misubishi_Packet_Manager.TcDUT
TYPE ST_Robot_Misubishi_Packet_Manager :
STRUCT
	StatusPacket					: ST_Robot_Mitsubishi_Packet_1000;								// Robot status packet structure.
	RobotBaseForStationPacket		: ST_Robot_Mitsubishi_Packet_1100;
	PacketConfirmationPacket		: ST_Robot_Mitsubishi_Packet_1101;	
	ProgramCompletedPacket			: ST_Robot_Mitsubishi_Packet_1102;	
	DependencyConfirmedPacket		: ST_Robot_Mitsubishi_Packet_1103;
	
	SettingsPacket					: ST_Robot_Mitsubishi_Packet_2000;								// Robot control packet structure.
	ControlPacket					: ST_Robot_Mitsubishi_Packet_2010;
	StateConfirmationPacket				:ST_Robot_Mitsubishi_Packet_2018;								
END_STRUCT
END_TYPE

// NB!!!
// Use these directly - 
// case receivedPacket.0 OF
//		1000 : MEMSET(StatusPacket, receivedPacket, LEN(StatusPacket));
//		.
//		.
//		.
// endCase
//

// ---- POUs/Mitsubishi/DUT/E_Communication_Send_States.TcDUT
{attribute 'qualified_only'}
{attribute 'strict'}
TYPE E_Communication_Send_States :
(
	E_COM_SEND_PREPARE := 0,
	E_COM_SEND_START_SEND,
	E_COM_SEND_WAIT_SENT,
	E_COM_SEND_FINALIZE
);
END_TYPE

// ---- POUs/Mitsubishi/DUT/E_Robot_Mitsubishi_States.TcDUT
{attribute 'qualified_only'}
{attribute 'strict'}
TYPE E_Robot_Mitsubishi_States :
(
	STATE_OPERATIONAL := 10,
	STATE_START_PROGRAM,
	STATE_WAIT_PROGRAM_COMPLETED,
	STATE_START_STOP,
	STATE_WAIT_STOP,
	STATE_STOPPED,
	STATE_SET_END,
	STATE_WAIT_SET_END,
	STATE_WAITING_RESET,
	STATE_START_RESET,
	STATE_WAITING_RESET_COMPLETED,
	STATE_START_POWER_ON,
	STATE_WAIT_POWERED_ON,
	STATE_START_POWER_OFF,
	STATE_WAIT_POWERED_OFF,
	STATE_REQUEST_DEPENDENCY_CONFIRMATION,
	STATE_WAIT_DEPENDENCY_CONFIRMATION,
	STATE_START_TARGET_SPEED_OVERRIDE_CHANGE,
	STATE_START_TARGET_TRAYPOS_CHANGE,
	STATE_START_TARGET_PROGRAM_CHANGE,
	STATE_START_TARGET_PROGRAM,
	STATE_WAIT_PROGRAM_STARTED,
	STATE_TOGGLE_GRIPERA,
	STATE_TOGGLE_GRIPERB,
	STATE_ERROR_ROBOT,
	STATE_ERROR_STATE_MACHINE := 100
)DINT;
END_TYPE

// ---- POUs/Mitsubishi/DUT/ST_Robot_Mitsubishi.TcDUT
TYPE ST_Robot_Mitsubishi :
STRUCT
// INPUTS 	
	bReady							: BOOL;															// Is the robot ready for operation.
	bBusy							: BOOL;															// Is the robot operating.
	bError							: BOOL;															// Is the robot in an error state.
	bDisabled						: BOOL;															// Is the robot in a disabled state.	
	bPoweredOn						: BOOL;															// Is the robot powered on.
	bAutomaticMode					: BOOL;															// Is the robot in automatic mode - can work.
	bExecuting						: BOOL;															// Is the robot executing - in a cycle/program.
	bEnding							: BOOL;															// Is the robot ending a cycle/program.
	bProgramCompleted				: BOOL;															// Is the last started program completed.	
	bOnline							: BOOL;															// Is the TCP IP communication to the robot active.
	bGripperAPresent				: BOOL;
	bGripperBPresent				: BOOL;
// Statuses
	nCurrentState					: E_Robot_Mitsubishi_States;									// The current robot state ID if defined.
	nLastState						: E_Robot_Mitsubishi_States;									// The previous state of the robot.
	nLastErrorState					: E_Robot_Mitsubishi_States;									// The last state where an error had occured.
	nDependencyState				: DINT;															// The dependency state of the robot.
	nCurrentProgram					: DINT;															// The current robot program.
	nCurrentTrayPosition			: DINT;															// The current station to work with.
	nCurrentSpeed					: DINT;															// The current speed overdive.
	nCurrentProductID				: DINT;
	nCurrentGripperID				: DINT;															// The current gripper ID if selected.
	nCurrentTrayOrient				: DINT;
	nCurrentTargetProgram			: DINT;															// The target robot program.
	nCurrentTargetTrayPosition		: DINT;															// The target station to work with.
	nCurrentTargetSpeed				: DINT;															// The target speed overdive.
	nCurrentTargetProductID			: DINT;
	nCurrentTargetGripperID			: DINT;	
	nCurrentTargetTrayOrient		: DINT;	
		
	nLastReceivedPacketID			: DINT;															// The ID of the last packet received.
	bLastPacketConfirmed			: BOOL;		// Not Used													// Had the last sent packet been confirmed.
	
	// OUTPUTS
// Control
	bDoReset						: BOOL;															// Reset the robot controller.+
	bDoServoOn						: BOOL;															// Enable the robot controller.
	bDoServoOff						: BOOL;															// Disable the robot controller.
	bDoStepFwd						: BOOL;															// Execute next step if in step mode.
	bDoStepBwd						: BOOL;															// Return to the previous step if in step mode.
	bDoEnd							: BOOL;															// End the current program.
	bDoStop							: BOOL;															// Stop the currently selected program if executing.
	bDoStart						: BOOL;															// Start the currently selected program.
	bDoOpenGripperA					: BOOL;
	bDoCloseGripperA				: BOOL;
	bDoOpenGripperB					: BOOL;
	bDoCloseGripperB				: BOOL;														
	bDoStartProgram					: BOOL;
	bDoChangeTargetTrayPosition		: BOOL;															// Change the target station.
	bDoChangeTargetProgram			: BOOL;															// Change the target program.
	bDoChangeTargetSpeed			: BOOL;															// Change the target speed - direct.
	bDoChangeTargetCorrection		: BOOL;															// Change the target correction.
	bDoChangeTargetProductID		: BOOL;															// Change the target product ID.
	bDoConfirmDependency			: BOOL;															// Confirm the dependency state.
	bToggleEnable					: BOOL;		//Not Used											// Use to enable operation of the state machine.
	bToggleConnect					: BOOL;															// Use to start/stop the socket communication.
	
// Settings
	nTargetTrayPosition				: DINT;															// The station of interest to be worked with.
	nTargetProgram					: DINT;															// The program to be executed.
	nTargetSpeed					: DINT;															// The speed overdrive to be set.
	nTargetProductID				: DINT;															// The target product id.
	nTargetGripperID				: DINT;															// The target gripper id.
	nTargetTrayOrientation			: DINT;															// The target tray orient.

	nLastSentPacketID				: DINT;		// Not Used											// The id of the last sent packet to the robot.
	
	sRobotAddress					: T_IPv4Addr;														// The IPv4 address of the robot server.
	nRobotPort						: UDINT;														// The port of the robot server.
END_STRUCT
END_TYPE

// ---- GVLs/Consts.TcGVL
{attribute 'qualified_only'}
VAR_GLOBAL CONSTANT
	
        // Общи	константии за машината

		MAX_IO_POINTS 		: INT     := 512;          // Максимален брой на IO image 
		MAX_SYNC_STATIONS   : DINT    := 64;		   // Максимален брой на dependancy-та едновремено
		DEP_PASS            : INT     := 1;            // Използват се в dependencySync - чрез тези променливи
		SYNC_CONFIRM        : INT     := 2;            // се реализира възможността да има мн. sync-кове в един state
		NO_ERROR       		: DINT    := 0;			   // Станцията няма грешка
		MIN_AXIS_LEN		: REAL    := 500;          // Мин. дългина на оста на стакерите
		MIN_PALLET_SIZE     : REAL    := 10;           // Мин. дебелина на тара
		MAX_AXIS_POS        : INT     := 20;           // Макс. брой позиция за оста на стакер
		LOAD_PALLETS_STEP   : INT     := 4; 		   // По колко тари да местят при зареждане стакерите наведнъж
		PURGE_CYCLES        : INT     := 32;           // Макс. брой завъртания на масата на InC при PURGE 
		MAX_RECIPE          : DINT    := 15;           // Макс. брой рецепти с който може да се работи
		ROT_PALLET			: DINT    := 1;            // Тарата трябва да се ротира преди да се остави
		TRANS_PALLET	    : DINT    := 2;            // Тарата се транслира преди да се остави
		
		// Констанити за станцийте - всяка едана state машина трябва да ги има
		
		ST_NULL			    : DINT    := 0;            // Това състояние да НЕ се дефинира в стъпковите машини - презен цикъл		
		ST_START_UP        	: DINT    := 1;            // Състояние на старт - влиза се за един цикъл в него при старт
		ST_INIT			   	: DINT	  := 10;           // Първо състояние за инициализация
        ST_READY 		   	: DINT    := 20;           // Станцията е готова за работа - от тук започва работния цикъл
		ST_STOP				: DINT    := 30;           // Станцията е спряна
        ST_STEP_BLOCK      	: DINT    := 40;           // Състояние за стъпков режим 
		ST_EMG				: DINT	  := 50;           // Има активен safety стоп
		

		
		// Константи за dependensy
		
		NO_DEPENDENCY      : DINT     := 0;            //  Няма dependency към друга станция
		
		// Кoнстанти за data requests
		
        NO_REQUEST         : DINT      := 0;            // Текущият data request е изпълнен
		REQUEST_ERROR      : DINT      := 1337;         // Има някаква грешка с текущият data request
			
END_VAR

// ---- GVLs/DEBUG.TcGVL
{attribute 'qualified_only'}
VAR_GLOBAL
	
    ioDebugActive          : BOOL := FALSE;
	noErrors               : BOOL := FALSE;
 
	machinedClearDep   	   : BOOL := FALSE;
	machinedClearSync      : BOOL := FALSE;
	
	sLoadClearDep          : BOOL := FALSE;
	sLoadClearSync         : BOOL := FALSE;
	
	sUnloadClearDep        : BOOL := FALSE;
	sUnloadClearSync       : BOOL := FALSE;

    incCommClearDep   	   : BOOL := FALSE;
	incCommClearSync       : BOOL := FALSE;
	
	insertLoadClearDep     : BOOL := FALSE;
	insertLoadClearSync    : BOOL := FALSE;
	
	insertUnloadClearDep   : BOOL := FALSE;
	insertUnloadClearSync  : BOOL := FALSE;

	roboClearDep           : BOOL := FALSE;
	roboClearSync          : BOOL := FALSE;
	
END_VAR

// ---- GVLs/Global.TcGVL
{attribute 'qualified_only'}
VAR_GLOBAL
	
	// Входен и изходен масив за IO Image
	
	INPUT_IMAGE   	    AT %I* : ARRAY[0..Consts.MAX_IO_POINTS] OF BYTE;
    OUTPUT_IMAGE   	    AT %Q* : ARRAY[0..Consts.MAX_IO_POINTS] OF BYTE;

	commands         : controlCommands;       // главни команди
	purgeActive      : BOOL; 				  // има започнала purge процедура
	openDoors        : BOOL;                  // има отворени врети
	emgStop	         : BOOL; 				  // има натиснат EMG Stop
	emgStopSignal	 : BOOL; 				  // сингнал за EMG  Stop към всички станций
	machError	     : BOOL; 				  // в някоя станция има грешка
	startZumer       : BOOL;				  // звукова сигнализация
	recipe           : DINT;                  // избраната рецепта за работа
	sensorStatus     : BOOL;                  // в гнездото под инсъртър 2 има сензор за разтоварване  
	palletFail       : BOOL;                  // робота не е могъл да вземе или е изпуснал тара
	lStackLastPallet : BOOL; 				  // входният стакер няма повече палети
	robotSafe        : BOOL;                  // робота е на безопастно място при инициализация
	sensorOnIUnload  : BOOL;                  // има сензор в гнездото под изх. инсъртър
	purgeDoneIL      : BOOL;                  // PURGE процедурата е завършила - сигнализира вх. инсъртър
	purgeDoneIU      : BOOL;                  // PURGE процедурата е завършила - сигнализира изх. инсъртър
	gnLostDPPackets  : INT;                   // Не се ползва
	RobotEMG         : BOOL;
	RobotNoCom       : BOOL;
	emptyLoadPallet  : BOOL;
	
	
	

 //   INPUT_IMAGE   : ARRAY [0..Consts.MAX_IO_POINTS] OF BYTE; 
 //	 OUTPUT_IMAGE  : ARRAY [0..Consts.MAX_IO_POINTS] OF BYTE;

END_VAR

// ---- GVLs/Stations.TcGVL
{attribute 'qualified_only'}
VAR_GLOBAL
	
    
	sLoadImageIO    			 : stackerLoadImage;
	sLoadHmiIO      		 	 : stackerLoadIO;
	sLoadStBase      		     : stationBase  := (ToggleEnable := TRUE, AutoMode := TRUE);
	sLoadSettings				 : stackerLoadSettings;
	sLoadDrive 					 : ST_MotorBase := (TargetPrecision := 0.01);
	sLoadAxis                    : AXIS_REF_CiA402_ETC_CMMT_AS;
	
	sUnloadImageIO       		 : stackerUnLoadImage;
	sUnloadHmiIO           		 : stackerUnLoadIO;
	sUnloadStBase         		 : stationBase  := (ToggleEnable := TRUE, AutoMode := TRUE);
	sUnloadSettings				 : stackerUnloadSettings;
	sUnloadDrive  				 : ST_MotorBase := (TargetPrecision := 0.01);
	sUnloadAxis                  : AXIS_REF_CiA402_ETC_CMMT_AS;
	
    insertLoadImageIO     		 : inserterLoadImage;
	insertLoadHmiIO       		 : inserterLoadIO;
	insertLoadStBase      		 : stationBase  := (ToggleEnable := TRUE, AutoMode := TRUE);
	insertLoadData               : dataRequestCam;
	insertLoadSetting            : inserterLoadSettings;
	insertLoadDrive				 : ST_MotorBase := (TargetPrecision := 0.01);
	insertLoadAxis               : T_LM_Axis; 
	
	insertUnLoadImageIO     	 : inserterUnLoadImage;
	insertUnLoadHmiIO       	 : inserterUnLoadIO;
	insertUnLoadStBase      	 : stationBase  := (ToggleEnable := TRUE, AutoMode := TRUE);
	insertUnloadSetting          : inserterUnloadSettings;
	insertUnLoadDrive			 : ST_MotorBase := (TargetPrecision := 0.01);
	insertUnLoadAxis             : T_LM_Axis; 
	
	roboImageIO         		 : roboArmImage;
	roboHmiIO                    : roboArmIO;
	roboStBase                   : stationBase := (ToggleEnable := TRUE, AutoMode := TRUE);
	roboSetings                  : roboArmSettings;
	roboData                     : dataRequestRobot;
	
	incCommImageIO         		 : incCommImage;
	incCommHmiIO                 : incCommIO;
	incCommStBase                : stationBase := (ToggleEnable := TRUE, AutoMode := TRUE);
	
	machineImageIO         		 : machineImage;
	machineHmiIO	             : machineIO;
	machineStBase                : stationBase := (ToggleEnable := TRUE, AutoMode := TRUE);	
	
	//======================================== Robot====================================================
	gstRobotMitsubishi: ST_Robot_Mitsubishi := (												
		nRobotPort := 10004,					// nRobotPort := 10004,
		bToggleEnable := TRUE,
		bToggleConnect := FALSE,
		bDoServoOn := FALSE,
		bDoReset := FALSE,
		nTargetTrayPosition := 0,
		nTargetProgram := 1,
		nTargetSpeed := 90,
		nTargetCorrectionID := 0,
		bLastPacketConfirmed := TRUE);																	// Robot Mitsubishi station.	
	gstRobotMitsubishiPacketManager	: ST_Robot_Misubishi_Packet_Manager;
    
	

END_VAR

// ---- GVLs/TagsHMI.TcGVL
{attribute 'qualified_only'}
VAR_GLOBAL
	
	   // Пишат се от HMI, четат се от TwinCat
		stopZumer      				: BOOL;          	// Сприране на сигнализация (има сигнализация при последна тара в Load Stacker)
		startPurge                  : BOOL;             // Стартирене на PURGE проседура на машаната
		camResult                   : DINT;             // Резултат от камерата
		
		// Пишат се от TwinCat, четат се от HMI
		AlarmActive                 : BOOL;             // Има активна аларма
		LoadStackerSignal           : BOOL;             // Входният стакер има нужда да се зареди с тари
		UnloadStackerSignal         : BOOL; 			// Изходният стакер има нужда да се зареди с тари 

		// Нови
		activeEmg                   : BOOL;
		doorsOpen                   : BOOL;
		noAir                       : BOOL;
		robotEmgActive              : BOOL;
		robotNoCom                  : BOOL;
		robotError                  : BOOL;
		
		// Ще ги обсъдим
		manualStackerLoad           : BOOL;
		manualStackerUnload         : BOOL;
		manualInserterLoad          : BOOL;
		manualInserterUnload        : BOOL;
		manualRobot                 : BOOL;
		manualMachine               : BOOL;

END_VAR

// ---- GVLs/TagsRobot.TcGVL
{attribute 'qualified_only'}
VAR_GLOBAL
	
        // Параметри за работа на робота
		
		roboRecipeNum               : DINT;             // Текущата рецепта с която роботa трябва да работи
		loadPalletPos				: DINT;             // Гнездо във входата тара над което трябва да иде робота
		unLoadPalletPos				: DINT;             // Гнездо в изходната тара над което трябва да иде робота	
		rotPallet                   : DINT;             // Необходимо ли е да се завърти тарата на определен ъгъл при взимане от LoadStacker
		loadPalletRot 			    : DINT;
		unLoadPallerRot             : DINT;
		
		robotComOnline 			    : BOOL;
		robotError                  : BOOL;
		
END_VAR

// ---- POUs/MAIN.TcPOU
PROGRAM MAIN
VAR
	
	machineCycle        : machineStation;
	incCommCycle		: incCommStation;
	stackerLoadCycle    : stackerLoadStation;
	stackerUnloadCycle  : stackerUnloadStation;
	insertLoadCycle     : insertLoadStation;
	insertUnloadCycle   : insertUnloadStation;
	roboArmCycle        : roboArmStation;

END_VAR




	machineCycle	   (stBase := Stations.machineStBase,      activeEMG := FALSE,                ioImage := Stations.machineImageIO,
				  		depClear:= DEBUG.machinedClearDep,     syncClear := DEBUG.machinedClearSync);
				
	incCommCycle	   (stBase := Stations.incCommStBase,      activeEMG := Global.emgStopSignal, ioImage := Stations.incCommImageIO,
				        depClear:= DEBUG.incCommClearDep,      syncClear := DEBUG.incCommClearSync);
				 
	stackerLoadCycle   (stBase := Stations.sLoadStBase,        activeEMG := Global.emgStopSignal, ioImage := Stations.sLoadImageIO,
				        depClear:= DEBUG.sLoadClearDep,        syncClear := DEBUG.sLoadClearSync);
				  
	stackerUnloadCycle (stBase := Stations.sUnloadStBase,      activeEMG := Global.emgStopSignal, ioImage := Stations.sUnloadImageIO,
				        depClear:= DEBUG.sUnloadClearDep,      syncClear := DEBUG.sUnloadClearSync);
					
	insertLoadCycle    (stBase := Stations.insertLoadStBase,   activeEMG := Global.emgStopSignal, ioImage := Stations.insertLoadImageIO,
				        depClear:= DEBUG.insertLoadClearDep,   syncClear := DEBUG.insertLoadClearSync);
					
	insertUnloadCycle  (stBase := Stations.insertUnloadStBase, activeEMG := Global.emgStopSignal, ioImage := Stations.insertUnLoadImageIO,
				        depClear:= DEBUG.insertUnloadClearDep, syncClear := DEBUG.insertUnloadClearSync);
					
	roboArmCycle       (stBase := Stations.roboStBase,         activeEMG := Global.emgStopSignal, ioImage := Stations.roboImageIO,
				       depClear:= DEBUG.roboClearDep,          syncClear := DEBUG.roboClearSync);

END_PROGRAM

// ---- POUs/Stations/machineStation.TcPOU
FUNCTION_BLOCK machineStation EXTENDS stateMachine
VAR_INPUT
	
	ioImage      : machineImage;

END_VAR
VAR
	
	activeState 	: machineStates;
	
	resetTime   	: TIME := T#2S;           // Време за ресет след ативиране на EMG stop
	resetSig		: BOOL := FALSE; 
	resetTimer		: TON;
	commandReady	: BOOL; 				  // Има приета нова команда
	errorPuls 		: R_TRIG;			      // Има нова грешка в машината
	
	purgeIndexDone  : BOOL := FALSE; 		  // Изчаква да се извадят всички бройки от масата
	purgeRobotDone  : BOOL := FALSE; 		  // Робота е приключил работа
	purgeStackers   : BOOL := FALSE;          // Стакерите са извадили всички тари от тях
	
	startZumer			   : BOOL;									   // Упр. на сигнален зумер
	zumerTimer1			   : TON;
	zumerTimer2			   : TON;
	zumerTimer3			   : TON;
	zumerBeep			   : INT;

END_VAR
VAR // added by the converter: edge detectors and wires of the graphical bodies
    _w1, _w2, _w3 : BOOL;
END_VAR


// Има разлики спрямо останалите станций на машита
// Някой states липсват и не може тази станция да минава в stop режим

zumer();                  // Упр. на сигният зумер

// Сигнали за HMI

	TagsHMI.activeEmg       := io.getX(ioImage.xEmgBnt);
	TagsHMI.doorsOpen       := io.getX(ioImage.xDoors);         
	TagsHMI.noAir           := io.getX(ioImage.xAirOk);            
	TagsHMI.robotEmgActive  := io.getX(ioImage.xRobotEmgOk);               
	TagsHMI.robotError      := TagsRobot.robotError;    


errorPuls(CLK := Global.machError); 

IF NOT io.getX(ioImage.xDoors) AND io.getX(ioImage.xAirOk) AND io.getX(ioImage.xEmgBnt) THEN
	Global.openDoors := TRUE;						// Има отворена вратa
	Global.emgStop   := FALSE;
	setDisplayState(machineDisplayStates.dStOpenDoors);
	setEmg(emgOrAlarm := TRUE);
	
ELSIF NOT io.getX(ioImage.xEmgBnt) THEN
	Global.emgStop   := TRUE; 					   //  Авариен стоп
	Global.openDoors := FALSE;	
	setDisplayState(machineDisplayStates.dStEMGButtonDown);
	setEmg(emgOrAlarm := TRUE);
	
ELSIF NOT io.getX(ioImage.xAirOk)  THEN
 	Global.emgStop   := TRUE; 					   // Няма оперативно налягане на въздуха   
	Global.openDoors := FALSE;	
	setDisplayState(machineDisplayStates.dStNoAirSupplay);
	setEmg(emgOrAlarm := TRUE);	
	
END_IF

IF NOT io.getX(ioImage.xRobotEmgOk)  THEN
 	Global.emgStop   := TRUE; 	                   //  Авариен стоп  на робота
	Global.RobotEMG  := TRUE;				      
	setDisplayState(machineDisplayStates.dStMachineRobotEMG);
	setEmg(emgOrAlarm := TRUE);		
END_IF

IF errorPuls.Q THEN
	setEmg(emgOrAlarm := FALSE);	
	Global.startZumer := TRUE;
END_IF

setStateVars(ioImage, activeState);


CASE activeState OF 
	
//  *** Start Up
//  Старт на станцията след подаване на захр.

